(* IEC 61131-3 sources: std_i2980_v2.06_cp053/Source/IMM/ieccontrol/GlobalBaseArchives (part 20) *)

(* ---- ABUpdateRelLintabPreInject.pu ---- *)
IMPORT_OVER_LISTFILE
 FFixCylinderData
, FCalculateCylinderSize
, FCalcScrewSize
, KAPPL_LintabData
, tsCylinderData
, FBDebugTrace

END_IMPORT

ALGORITHM_BLOCK ABUpdateRelLintabPreInject #DUMMY_EDIT_BLOCK

SYSTEM_VAR
 sv_bCalcMaxValuesFromCylData : BOOL (* TRUE: calculate max speed and max pressure values by using cylinder data;  FALSE: max values must be entered manually *);
END_VAR

SYSTEM_OBJECT
 PU_Task_7 : TASK;
END_OBJECT

VAR
 mpLintabOut : REFTO KAPPL_LintabData;
 mpCylinderData : REFTO tsCylinderData;
 mprMaxPressure : REFTO REAL;
 mprMaxHydrPressure : REFTO REAL;
 mbInitDone : BOOL;
 mprScrewDiameter : REFTO REAL;
END_VAR

ALGORITHM aUpdateLintabOut

#BEGIN_EDIT_BLOCK
(**************************************** WARNING ********************************************
 *** The KEBA Kemro K2 System including software is not intended for safety control tasks! ***
 ***                       For further information see Comment tab!                        ***
 *********************************************************************************************)

// save data to Pre lintab
// normally a 1:1 lintab
mpLintabOut^.LintabPoints.uNoOfPoints := 2;
mpLintabOut^.LintabPoints.Point[1].rX := 0.0;
mpLintabOut^.LintabPoints.Point[1].rY := 0.0;
mpLintabOut^.LintabPoints.Point[2].rX := mprMaxPressure^;
mpLintabOut^.LintabPoints.Point[2].rY := mprMaxHydrPressure^;

;#END_EDIT_BLOCK END_ALGORITHM

ALGORITHM aCalcMaxPressure

VAR_TEMP
 rCylinderSize : REAL (* size of cylinder im mm˛ *);
 rScrewSize : REAL (* size of screw in mm˛ *);
 tmp : BOOL;
END_VAR
#BEGIN_EDIT_BLOCK
(**************************************** WARNING ********************************************
 *** The KEBA Kemro K2 System including software is not intended for safety control tasks! ***
 ***                       For further information see Comment tab!                        ***
 *********************************************************************************************)

IF NOT sv_bCalcMaxValuesFromCylData THEN
   // no calculation necessary
   RETURN;
END_IF;

tmp := FFixCylinderData(mpCylinderData);

// sanity check
IF mprScrewDiameter^ <= 0.0 THEN
   mprScrewDiameter^ := 34.0;
END_IF;

rCylinderSize := FCalculateCylinderSize(CylinderData := mpCylinderData^, bSmallSize := mpCylinderData^.bUseSmallSize,bCalcHighPressSize := FALSE);

rScrewSize := FCalcScrewSize(mprScrewDiameter^);

// calculate pressure for screw
mprMaxPressure^ := mprMaxHydrPressure^ * rCylinderSize / rScrewSize;

;#END_EDIT_BLOCK END_ALGORITHM

ALGORITHM aInit

VAR_INPUT
 pLintabOut : REFTO KAPPL_LintabData;
 prMaxPressure : REFTO REAL (* reference to calculated max. pressure *);
 prMaxHydrPressure : REFTO REAL (* reference to max. possible hydraulic pressure (depends on used pumps(s)) *);
 pCylinderData : REFTO tsCylinderData;
 prScrewDiameter : REFTO REAL (* diameter of screw in mm *);
END_VAR

VAR
 fbDebugTrace : FBDebugTrace;
END_VAR
#BEGIN_EDIT_BLOCK
(**************************************** WARNING ********************************************
 *** The KEBA Kemro K2 System including software is not intended for safety control tasks! ***
 ***                       For further information see Comment tab!                        ***
 *********************************************************************************************)

mbInitDone := FALSE;
mpCylinderData := pCylinderData;
mpLintabOut := pLintabOut;
mprMaxPressure := prMaxPressure;
mprMaxHydrPressure := prMaxHydrPressure;
mprScrewDiameter := prScrewDiameter;

IF NOT CHECK_REF(pCylinderData^) THEN
   fbDebugTrace('pCylinderData not valid');
   RETURN;
END_IF;

IF (NOT CHECK_REF(prScrewDiameter^)) THEN
   fbDebugTrace('prScrewDiameter not valid');
   RETURN;
END_IF;

IF (NOT CHECK_REF(pLintabOut^)) THEN
   fbDebugTrace('pLintabOut not valid');
   RETURN;
END_IF;

IF (NOT CHECK_REF(prMaxPressure^)) THEN
   fbDebugTrace('prMaxPressure not valid');
   RETURN;
END_IF;

IF (NOT CHECK_REF(prMaxHydrPressure^)) THEN
   fbDebugTrace('prMaxHydrPressure not valid');
   RETURN;
END_IF;

// init successful
mbInitDone := TRUE;

aCalcMaxPressure();

aUpdateLintabOut();

;#END_EDIT_BLOCK END_ALGORITHM

POSTUPDATE_ALGORITHM pUpdatePressure ON PU_Task_7 WITH mprMaxHydrPressure^,mpCylinderData^,mprScrewDiameter^

#BEGIN_EDIT_BLOCK
(**************************************** WARNING ********************************************
 *** The KEBA Kemro K2 System including software is not intended for safety control tasks! ***
 ***                       For further information see Comment tab!                        ***
 *********************************************************************************************)

IF NOT mbInitDone THEN
    RETURN;
END_IF;

aCalcMaxPressure();

;#END_EDIT_BLOCK END_ALGORITHM

POSTUPDATE_ALGORITHM pUpdatePressureLintab ON PU_Task_7 WITH mprMaxHydrPressure^,mprMaxPressure^

#BEGIN_EDIT_BLOCK
(**************************************** WARNING ********************************************
 *** The KEBA Kemro K2 System including software is not intended for safety control tasks! ***
 ***                       For further information see Comment tab!                        ***
 *********************************************************************************************)

IF NOT mbInitDone THEN
    RETURN;
END_IF;

// update lintab
aUpdateLintabOut();

;#END_EDIT_BLOCK END_ALGORITHM

END_ALGORITHM_BLOCK

#END_OF_IEC_PART

@Puma @IecEditor 6 114 @Pou 25
@@@BEG_Comment@@@

@@@END_Comment@@@

@BEG_Contents

@BEG_Func
@RT(17)FuncTreeContainer
3
@Var @RT(16)FFixCylinderData @RT(0) @T @T @DERIVED 0 @F @RT(8)FUNCTION @F
@T
@BEG_Attrib
0 @RT(0) @RT(0)
@END_Attrib
1 1 @F @F @F @F

@Var @RT(22)FCalculateCylinderSize @RT(0) @T @T @DERIVED 0 @F @RT(8)FUNCTION @F
@T
@BEG_Attrib
0 @RT(0) @RT(0)
@END_Attrib
1 1 @F @F @F @F

@Var @RT(14)FCalcScrewSize @RT(0) @T @T @DERIVED 0 @F @RT(8)FUNCTION @F
@T
@BEG_Attrib
0 @RT(0) @RT(0)
@END_Attrib
1 1 @F @F @F @F

@END_Func

@BEG_Const
@RT(18)ConstTreeContainer
0
@END_Const

@BEG_Export

@BEG_Kind
@ALGORITHM_BLOCK @RT(26)ABUpdateRelLintabPreInject @STRUCTURED_TEXT
@RT(0) @RT(0) @RT(0)
@END_Kind

@BEG_Dcl
@RT(16)DclTreeContainer
8
@Var @RT(28)sv_bCalcMaxValuesFromCylData @RT(0) @T @F @DT @RT(4)BOOL @RT(0) @T @T @BASIC 0 @F
@F @F
@T
@BEG_Attrib
3 @RT(0) @RT(117)TRUE: calculate max speed and max pressure values by using cylinder data;  FALSE: max values must be entered manually @RT(0)
@END_Attrib
1 8 @F @F @F @F

@Var @RT(9)PU_Task_7 @RT(0) @T @F @DT @RT(4)TASK @RT(0) @T @T @BASIC 0 @F
@F @F
@T
@BEG_Attrib
3 @RT(0) @RT(0) @RT(0)
@END_Attrib
1 7 @F @F @F @F

@Var @RT(11)mpLintabOut @RT(0) @T @T @REFTO 0 @F @DERIVED 0 @T @T @DT @RT(16)KAPPL_LintabData @RT(0) @T @T @UNKNOWN 0 @F
@F @F
@T
@BEG_Attrib
3 @RT(0) @RT(0) @RT(0)
@END_Attrib
1 0 @F @F @F @F

@Var @RT(14)mpCylinderData @RT(0) @T @T @REFTO 0 @F @DERIVED 0 @T @T @DT @RT(14)tsCylinderData @RT(0) @T @T @UNKNOWN 0 @F
@F @F
@T
@BEG_Attrib
3 @RT(0) @RT(0) @RT(0)
@END_Attrib
1 0 @F @F @F @F

@Var @RT(14)mprMaxPressure @RT(0) @T @T @REFTO 0 @T @DT @RT(4)REAL @RT(0) @T @T @BASIC 0 @F
@F @F
@T
@BEG_Attrib
3 @RT(0) @RT(0) @RT(0)
@END_Attrib
1 0 @F @F @F @F

@Var @RT(18)mprMaxHydrPressure @RT(0) @T @T @REFTO 0 @T @DT @RT(4)REAL @RT(0) @T @T @BASIC 0 @F
@F @F
@T
@BEG_Attrib
3 @RT(0) @RT(0) @RT(0)
@END_Attrib
1 0 @F @F @F @F

@Var @RT(10)mbInitDone @RT(0) @T @F @DT @RT(4)BOOL @RT(0) @T @T @BASIC 0 @F
@F @F
@T
@BEG_Attrib
3 @RT(0) @RT(0) @RT(0)
@END_Attrib
1 0 @F @F @F @F

@Var @RT(16)mprScrewDiameter @RT(0) @T @T @REFTO 0 @T @DT @RT(4)REAL @RT(0) @T @T @BASIC 0 @F
@F @F
@T
@BEG_Attrib
3 @RT(0) @RT(0) @RT(0)
@END_Attrib
1 0 @F @F @F @F

@END_Dcl

@END_Export

@BEG_Body

5

@BEG_Export

@BEG_Algo
@ALGORITHM @RT(16)aUpdateLintabOut @STRUCTURED_TEXT
@RT(0) @RT(0) @RT(0) @F @F
@END_Algo

@BEG_Dcl
@RT(16)DclTreeContainer
0
@END_Dcl

@END_Export

@BEG_Export

@BEG_Algo
@ALGORITHM @RT(16)aCalcMaxPressure @STRUCTURED_TEXT
@RT(0) @RT(0) @RT(0) @F @F
@END_Algo

@BEG_Dcl
@RT(16)DclTreeContainer
3
@Var @RT(13)rCylinderSize @RT(0) @T @F @DT @RT(4)REAL @RT(0) @T @T @BASIC 0 @F
@F @F
@T
@BEG_Attrib
3 @RT(0) @RT(23)size of cylinder im mm˛ @RT(0)
@END_Attrib
1 4 @F @F @F @F

@Var @RT(10)rScrewSize @RT(0) @T @F @DT @RT(4)REAL @RT(0) @T @T @BASIC 0 @F
@F @F
@T
@BEG_Attrib
3 @RT(0) @RT(20)size of screw in mm˛ @RT(0)
@END_Attrib
1 4 @F @F @F @F

@Var @RT(3)tmp @RT(0) @T @F @DT @RT(4)BOOL @RT(0) @T @T @BASIC 0 @F
@F @F
@T
@BEG_Attrib
3 @RT(0) @RT(0) @RT(0)
@END_Attrib
1 4 @F @F @F @F

@END_Dcl

@END_Export

@BEG_Export

@BEG_Algo
@ALGORITHM @RT(5)aInit @STRUCTURED_TEXT
@RT(0) @RT(0) @RT(0) @F @F
@END_Algo

@BEG_Dcl
@RT(16)DclTreeContainer
6
@Var @RT(10)pLintabOut @RT(0) @T @T @REFTO 0 @F @DERIVED 0 @T @T @DT @RT(16)KAPPL_LintabData @RT(0) @T @T @UNKNOWN 0 @F
@F @F
@T
@BEG_Attrib
3 @RT(0) @RT(0) @RT(0)
@END_Attrib
1 1 @F @F @F @F

@Var @RT(13)prMaxPressure @RT(0) @T @T @REFTO 0 @T @DT @RT(4)REAL @RT(0) @T @T @BASIC 0 @F
@F @F
@T
@BEG_Attrib
3 @RT(0) @RT(37)reference to calculated max. pressure @RT(0)
@END_Attrib
1 1 @F @F @F @F

@Var @RT(17)prMaxHydrPressure @RT(0) @T @T @REFTO 0 @T @DT @RT(4)REAL @RT(0) @T @T @BASIC 0 @F
@F @F
@T
@BEG_Attrib
3 @RT(0) @RT(72)reference to max. possible hydraulic pressure (depends on used pumps(s)) @RT(0)
@END_Attrib
1 1 @F @F @F @F

@Var @RT(13)pCylinderData @RT(0) @T @T @REFTO 0 @F @DERIVED 0 @T @T @DT @RT(14)tsCylinderData @RT(0) @T @T @UNKNOWN 0 @F
@F @F
@T
@BEG_Attrib
3 @RT(0) @RT(0) @RT(0)
@END_Attrib
1 1 @F @F @F @F

@Var @RT(15)prScrewDiameter @RT(0) @T @T @REFTO 0 @T @DT @RT(4)REAL @RT(0) @T @T @BASIC 0 @F
@F @F
@T
@BEG_Attrib
3 @RT(0) @RT(23)diameter of screw in mm @RT(0)
@END_Attrib
1 1 @F @F @F @F

@Var @RT(12)fbDebugTrace @RT(0) @T @T @DERIVED 0 @F @RT(12)FBDebugTrace @F
@T
@BEG_Attrib
3 @RT(0) @RT(0) @RT(0)
@END_Attrib
1 0 @F @F @F @F

@END_Dcl

@END_Export

@BEG_Export

@BEG_Algo
@POSTUPDATE_ALGORITHM @RT(15)pUpdatePressure @STRUCTURED_TEXT
@RT(0) @RT(53)mprMaxHydrPressure^,mpCylinderData^,mprScrewDiameter^ @RT(9)PU_Task_7 @F @F
@END_Algo

@BEG_Dcl
@RT(16)DclTreeContainer
0
@END_Dcl

@END_Export

@BEG_Export

@BEG_Algo
@POSTUPDATE_ALGORITHM @RT(21)pUpdatePressureLintab @STRUCTURED_TEXT
@RT(0) @RT(35)mprMaxHydrPressure^,mprMaxPressure^ @RT(9)PU_Task_7 @F @F
@END_Algo

@BEG_Dcl
@RT(16)DclTreeContainer
0
@END_Dcl

@END_Export

@BEG_Body
@TL(13)
(**************************************** WARNING ********************************************
 *** The KEBA Kemro K2 System including software is not intended for safety control tasks! ***
 ***                       For further information see Comment tab!                        ***
 *********************************************************************************************)

// save data to Pre lintab
// normally a 1:1 lintab
mpLintabOut^.LintabPoints.uNoOfPoints := 2;
mpLintabOut^.LintabPoints.Point[1].rX := 0.0;
mpLintabOut^.LintabPoints.Point[1].rY := 0.0;
mpLintabOut^.LintabPoints.Point[2].rX := mprMaxPressure^;
mpLintabOut^.LintabPoints.Point[2].rY := mprMaxHydrPressure^;

@END_Body

@@@BEG_Comment@@@
@TL(0)

@@@END_Comment@@@

@BEG_Body
@TL(25)
(**************************************** WARNING ********************************************
 *** The KEBA Kemro K2 System including software is not intended for safety control tasks! ***
 ***                       For further information see Comment tab!                        ***
 *********************************************************************************************)

IF NOT sv_bCalcMaxValuesFromCylData THEN
   // no calculation necessary
   RETURN;
END_IF;

tmp := FFixCylinderData(mpCylinderData);

// sanity check
IF mprScrewDiameter^ <= 0.0 THEN
   mprScrewDiameter^ := 34.0;
END_IF;

rCylinderSize := FCalculateCylinderSize(CylinderData := mpCylinderData^, bSmallSize := mpCylinderData^.bUseSmallSize,bCalcHighPressSize := FALSE);

rScrewSize := FCalcScrewSize(mprScrewDiameter^);

// calculate pressure for screw
mprMaxPressure^ := mprMaxHydrPressure^ * rCylinderSize / rScrewSize;

@END_Body

@@@BEG_Comment@@@
@TL(0)

@@@END_Comment@@@

@BEG_Body
@TL(45)
(**************************************** WARNING ********************************************
 *** The KEBA Kemro K2 System including software is not intended for safety control tasks! ***
 ***                       For further information see Comment tab!                        ***
 *********************************************************************************************)

mbInitDone := FALSE;
mpCylinderData := pCylinderData;
mpLintabOut := pLintabOut;
mprMaxPressure := prMaxPressure;
mprMaxHydrPressure := prMaxHydrPressure;
mprScrewDiameter := prScrewDiameter;

IF NOT CHECK_REF(pCylinderData^) THEN
   fbDebugTrace('pCylinderData not valid');
   RETURN;
END_IF;

IF (NOT CHECK_REF(prScrewDiameter^)) THEN
   fbDebugTrace('prScrewDiameter not valid');
   RETURN;
END_IF;

IF (NOT CHECK_REF(pLintabOut^)) THEN
   fbDebugTrace('pLintabOut not valid');
   RETURN;
END_IF;

IF (NOT CHECK_REF(prMaxPressure^)) THEN
   fbDebugTrace('prMaxPressure not valid');
   RETURN;
END_IF;

IF (NOT CHECK_REF(prMaxHydrPressure^)) THEN
   fbDebugTrace('prMaxHydrPressure not valid');
   RETURN;
END_IF;

// init successful
mbInitDone := TRUE;

aCalcMaxPressure();

aUpdateLintabOut();

@END_Body

@@@BEG_Comment@@@
@TL(0)

@@@END_Comment@@@

@BEG_Body
@TL(11)
(**************************************** WARNING ********************************************
 *** The KEBA Kemro K2 System including software is not intended for safety control tasks! ***
 ***                       For further information see Comment tab!                        ***
 *********************************************************************************************)

IF NOT mbInitDone THEN
    RETURN;
END_IF;

aCalcMaxPressure();

@END_Body

@@@BEG_Comment@@@
@TL(0)

@@@END_Comment@@@

@BEG_Body
@TL(12)
(**************************************** WARNING ********************************************
 *** The KEBA Kemro K2 System including software is not intended for safety control tasks! ***
 ***                       For further information see Comment tab!                        ***
 *********************************************************************************************)

IF NOT mbInitDone THEN
    RETURN;
END_IF;

// update lintab
aUpdateLintabOut();

@END_Body

@@@BEG_Comment@@@
@TL(0)

@@@END_Comment@@@
@END_Body

@END_Contents

(* ---- ABUpdateRelLintabVel.pu ---- *)
IMPORT_OVER_LISTFILE
 FFixCylinderData
, FCalculateCylinderSize
, FScaleAndFloor
, tnDataState
, KAPPL_LintabData
, tsCylinderData

END_IMPORT

ALGORITHM_BLOCK ABUpdateRelLintabVel #DUMMY_EDIT_BLOCK

SYSTEM_VAR
 sv_bCalcMaxValuesFromCylData : BOOL (* TRUE: calculate max speed and max pressure values by using cylinder data;  FALSE: max values must be entered manually *);
 sv_DataState : tnDataState;
 sv_iReadMachineDataCount : UDINT;
END_VAR

SYSTEM_OBJECT
 PU_Task_7 : TASK;
 PU_Task_3 : TASK;
END_OBJECT

VAR
 mpLintabOut : REFTO KAPPL_LintabData (* OUT: velocity lintab of movement *);
 mprAbsFlow : REFTO REAL (* IN: maximum absolute flow in l/min *);
 mpCylinderData : REFTO tsCylinderData (* IN: cylinder data *);
 mprMaxSpeed : REFTO REAL (* IN/OUT: max speed of movement *);
 mprMaxSpeedCalc : REFTO REAL (* IN/OUT: max speed of movement (calculated) *);
 mprMaxSpeedCalib : REFTO REAL (* IN/OUT: max speed of movement (calculated) *);
 mbprMaxSpeedCalibLinked : BOOL := FALSE (* IN/OUT: max speed of movement (calculated) *);
 mprMaxSpeedReducePercent : REFTO REAL (* IN: percentage to reduce max speed *);
 miMaxSpeedDigitsToFloor : SINT := 0 (* IN: max speed digits to floor *);
 mbInitDone : BOOL;
 mbFwd : BOOL;
END_VAR

ALGORITHM aUpdateLintabOut

#BEGIN_EDIT_BLOCK
(**************************************** WARNING ********************************************
 *** The KEBA Kemro K2 System including software is not intended for safety control tasks! ***
 ***                       For further information see Comment tab!                        ***
 *********************************************************************************************)

// save data to Vel lintab
mpLintabOut^.LintabPoints.uNoOfPoints := 2;
mpLintabOut^.LintabPoints.Point[1].rX := 0.0;
mpLintabOut^.LintabPoints.Point[1].rY := 0.0;
mpLintabOut^.LintabPoints.Point[2].rX := mprMaxSpeedCalc^;
mpLintabOut^.LintabPoints.Point[2].rY := 100.0; // %

;#END_EDIT_BLOCK END_ALGORITHM

ALGORITHM aCalcMaxVelocity

VAR_TEMP
 tmp : BOOL;
END_VAR

VAR
 rMaxFlow : REAL (* maximum flow in mm^3/sec *);
 rSize : REAL;
 bSmallSize : BOOL;
 rScalePercent : REAL;
END_VAR
#BEGIN_EDIT_BLOCK
(**************************************** WARNING ********************************************
 *** The KEBA Kemro K2 System including software is not intended for safety control tasks! ***
 ***                       For further information see Comment tab!                        ***
 *********************************************************************************************)

IF NOT sv_bCalcMaxValuesFromCylData THEN
   // no calculation necessary
   RETURN;
END_IF;

tmp := FFixCylinderData(mpCylinderData);

// convert from l/min to mm^3/sec
rMaxFlow := mprAbsFlow^ * 100.0 *100.0 *100.0 / 60.0;

bSmallSize := mbFwd AND mpCylinderData^.bUseSmallSize OR
                 ((NOT mbFwd AND NOT mpCylinderData^.bUseSmallSize));

rSize := FCalculateCylinderSize(CylinderData := mpCylinderData^,
                                bSmallSize := bSmallSize,
                                bCalcHighPressSize := FALSE);
// mmł/s / mm˛ ->mm/s
mprMaxSpeedCalc^ := rMaxFlow / rSize;
IF ((mbInitDone AND sv_DataState = nReady) AND (mprMaxSpeed^ > mprMaxSpeedCalc^)) THEN
   // prevent recalculation on machine data load except if max. value exceeds custom value
   rScalePercent := 100.0;
   IF mprMaxSpeedReducePercent <> EMPTY THEN
      rScalePercent := 100.0 - mprMaxSpeedReducePercent^;
   END_IF;
   mprMaxSpeed^ := FScaleAndFloor(mprMaxSpeedCalc^, rScalePercent, miMaxSpeedDigitsToFloor);
END_IF;
// check max velocity for visualization
IF (mbprMaxSpeedCalibLinked) THEN
   IF(mprMaxSpeedCalib^ <= 0.0) OR (mprMaxSpeedCalib^ > mprMaxSpeedCalc^) THEN
      mprMaxSpeedCalib^ := mprMaxSpeedCalc^;
   END_IF;
END_IF;

;#END_EDIT_BLOCK END_ALGORITHM

ALGORITHM aInit

VAR_INPUT
 pLintabOut : REFTO KAPPL_LintabData;
 prMaxSpeed : REFTO REAL;
 prMaxSpeedCalc : REFTO REAL;
 prAbsFlow : REFTO REAL (* absolute flow in l/min *);
 bFwd : BOOL (* TRUE if block is used for fwd movement *);
 pCylinderData : REFTO tsCylinderData;
 prMaxSpeedReducePercent : REFTO REAL;
 iMaxSpeedDigitsToFloor : SINT;
 prMaxSpeedCalib : REFTO REAL;
END_VAR

VAR
 // prMaxPumpFlow : REFTO REAL;
 tmp : DINT;
END_VAR
#BEGIN_EDIT_BLOCK
(**************************************** WARNING ********************************************
 *** The KEBA Kemro K2 System including software is not intended for safety control tasks! ***
 ***                       For further information see Comment tab!                        ***
 *********************************************************************************************)

mbInitDone := FALSE;
mprAbsFlow := prAbsFlow;
mpCylinderData := pCylinderData;
mpLintabOut := pLintabOut;
mprMaxSpeed := prMaxSpeed;
mprMaxSpeedCalc := prMaxSpeedCalc;
mprMaxSpeedCalib := prMaxSpeedCalib;
mprMaxSpeedReducePercent := prMaxSpeedReducePercent;
miMaxSpeedDigitsToFloor := iMaxSpeedDigitsToFloor;
mbFwd := bFwd;

IF NOT CHECK_REF(prAbsFlow^) THEN
    tmp := Print('prAbsFlow not valid');
    RETURN;
END_IF;

IF NOT CHECK_REF(pCylinderData^) THEN
    tmp := Print('pCylinderData not valid');
    RETURN;
END_IF;

IF (NOT CHECK_REF(pLintabOut^)) THEN
    tmp := Print('pLintabOut not valid');
    RETURN;
END_IF;

IF (NOT CHECK_REF(prMaxSpeed^)) THEN
    tmp := Print('prMaxSpeed not valid');
    RETURN;
END_IF;

IF (NOT CHECK_REF(prMaxSpeedCalc^)) THEN
    tmp := Print('prMaxSpeedCalc not valid');
    RETURN;
END_IF;

IF (CHECK_REF(mprMaxSpeedCalib^)) THEN
    mbprMaxSpeedCalibLinked := TRUE;
END_IF;

aCalcMaxVelocity();

//update lintab
aUpdateLintabOut();

// init successful
mbInitDone := TRUE;

;#END_EDIT_BLOCK END_ALGORITHM

POSTUPDATE_ALGORITHM pUpdateVelocity ON PU_Task_7 WITH mprAbsFlow^,mpCylinderData^

#BEGIN_EDIT_BLOCK
(**************************************** WARNING ********************************************
 *** The KEBA Kemro K2 System including software is not intended for safety control tasks! ***
 ***                       For further information see Comment tab!                        ***
 *********************************************************************************************)

IF NOT mbInitDone OR (sv_DataState = nReadMachineData) THEN
   RETURN;
END_IF;

// reset calib value if diameter or flow is changed
IF mbprMaxSpeedCalibLinked AND (sv_DataState = nReady) THEN
   mprMaxSpeedCalib^ := 0.0;
END_IF;

aCalcMaxVelocity();

;#END_EDIT_BLOCK END_ALGORITHM

POSTUPDATE_ALGORITHM pUpdateVelocityLintab ON PU_Task_7 WITH mprMaxSpeedCalc^

#BEGIN_EDIT_BLOCK
(**************************************** WARNING ********************************************
 *** The KEBA Kemro K2 System including software is not intended for safety control tasks! ***
 ***                       For further information see Comment tab!                        ***
 *********************************************************************************************)

IF NOT mbInitDone THEN
    RETURN;
END_IF;

aUpdateLintabOut();

;#END_EDIT_BLOCK END_ALGORITHM

POSTUPDATE_ALGORITHM pUpdateMaxVelocity ON PU_Task_7 WITH mprMaxSpeedCalib^

VAR
 rScalePercent : REAL;
END_VAR
#BEGIN_EDIT_BLOCK
(**************************************** WARNING ********************************************
 *** The KEBA Kemro K2 System including software is not intended for safety control tasks! ***
 ***                       For further information see Comment tab!                        ***
 *********************************************************************************************)

IF sv_DataState = nReadMachineData THEN
   RETURN;
END_IF;

IF ((mprMaxSpeedCalib^ < mprMaxSpeed^) AND (mprMaxSpeedCalib^ > 0.0)) THEN
   rScalePercent := 100.0;
   IF mprMaxSpeedReducePercent <> EMPTY THEN
      rScalePercent := 100.0 - mprMaxSpeedReducePercent^;
   END_IF;
   mprMaxSpeed^ := FScaleAndFloor(mprMaxSpeedCalib^, rScalePercent, miMaxSpeedDigitsToFloor);
END_IF;

;#END_EDIT_BLOCK END_ALGORITHM

POSTUPDATE_ALGORITHM pMachineDataLoaded ON PU_Task_7 WITH sv_iReadMachineDataCount

#BEGIN_EDIT_BLOCK
(**************************************** WARNING ********************************************
 *** The KEBA Kemro K2 System including software is not intended for safety control tasks! ***
 ***                       For further information see Comment tab!                        ***
 *********************************************************************************************)

aCalcMaxVelocity();

;#END_EDIT_BLOCK END_ALGORITHM

POSTUPDATE_ALGORITHM pMachineDataLoadingStarted ON PU_Task_3(1) WITH sv_DataState

#BEGIN_EDIT_BLOCK
(**************************************** WARNING ********************************************
 *** The KEBA Kemro K2 System including software is not intended for safety control tasks! ***
 ***                       For further information see Comment tab!                        ***
 *********************************************************************************************)

IF sv_DataState = nReadMachineData THEN
   //reset max speed calib at the beginning of machine data loading
   //if max speed calib is part of the loaded machine data, the correct value comes from the XMl file
   //if max speed calib is not part of machine data it is set to max speed calc
   //when calling aCalcMaxVelocity after loading machine data is finished
   IF mbprMaxSpeedCalibLinked THEN
      mprMaxSpeedCalib^ := 0.0;
   END_IF;
END_IF;

;#END_EDIT_BLOCK END_ALGORITHM

END_ALGORITHM_BLOCK

#END_OF_IEC_PART

@Puma @IecEditor 6 114 @Pou 25
@@@BEG_Comment@@@

@@@END_Comment@@@

@BEG_Contents

@BEG_Func
@RT(17)FuncTreeContainer
3
@Var @RT(16)FFixCylinderData @RT(0) @T @T @DERIVED 0 @F @RT(8)FUNCTION @F
@T
@BEG_Attrib
0 @RT(0) @RT(0)
@END_Attrib
1 1 @F @F @F @F

@Var @RT(22)FCalculateCylinderSize @RT(0) @T @T @DERIVED 0 @F @RT(8)FUNCTION @F
@T
@BEG_Attrib
0 @RT(0) @RT(0)
@END_Attrib
1 1 @F @F @F @F

@Var @RT(14)FScaleAndFloor @RT(0) @T @T @DERIVED 0 @F @RT(8)FUNCTION @F
@T
@BEG_Attrib
0 @RT(0) @RT(0)
@END_Attrib
1 1 @F @F @F @F

@END_Func

@BEG_Const
@RT(18)ConstTreeContainer
0
@END_Const

@BEG_Export

@BEG_Kind
@ALGORITHM_BLOCK @RT(20)ABUpdateRelLintabVel @STRUCTURED_TEXT
@RT(0) @RT(0) @RT(0)
@END_Kind

@BEG_Dcl
@RT(16)DclTreeContainer
16
@Var @RT(28)sv_bCalcMaxValuesFromCylData @RT(0) @T @F @DT @RT(4)BOOL @RT(0) @T @T @BASIC 0 @F
@F @F
@T
@BEG_Attrib
3 @RT(0) @RT(117)TRUE: calculate max speed and max pressure values by using cylinder data;  FALSE: max values must be entered manually @RT(0)
@END_Attrib
1 8 @F @F @F @F

@Var @RT(12)sv_DataState @RT(0) @T @T @DERIVED 0 @T @T @DT @RT(11)tnDataState @RT(0) @T @T @UNKNOWN 0 @F
@F @F
@T
@BEG_Attrib
3 @RT(0) @RT(0) @RT(0)
@END_Attrib
1 8 @F @F @F @F

@Var @RT(9)PU_Task_7 @RT(0) @T @F @DT @RT(4)TASK @RT(0) @T @T @BASIC 0 @F
@F @F
@T
@BEG_Attrib
3 @RT(0) @RT(0) @RT(0)
@END_Attrib
1 7 @F @F @F @F

@Var @RT(11)mpLintabOut @RT(0) @T @T @REFTO 0 @F @DERIVED 0 @T @T @DT @RT(16)KAPPL_LintabData @RT(0) @T @T @UNKNOWN 0 @F
@F @F
@T
@BEG_Attrib
3 @RT(0) @RT(32)OUT: velocity lintab of movement @RT(0)
@END_Attrib
1 0 @F @F @F @F

@Var @RT(10)mprAbsFlow @RT(0) @T @T @REFTO 0 @T @DT @RT(4)REAL @RT(0) @T @T @BASIC 0 @F
@F @F
@T
@BEG_Attrib
3 @RT(0) @RT(34)IN: maximum absolute flow in l/min @RT(0)
@END_Attrib
1 0 @F @F @F @F

@Var @RT(14)mpCylinderData @RT(0) @T @T @REFTO 0 @F @DERIVED 0 @T @T @DT @RT(14)tsCylinderData @RT(0) @T @T @UNKNOWN 0 @F
@F @F
@T
@BEG_Attrib
3 @RT(0) @RT(17)IN: cylinder data @RT(0)
@END_Attrib
1 0 @F @F @F @F

@Var @RT(11)mprMaxSpeed @RT(0) @T @T @REFTO 0 @T @DT @RT(4)REAL @RT(0) @T @T @BASIC 0 @F
@F @F
@T
@BEG_Attrib
3 @RT(0) @RT(29)IN/OUT: max speed of movement @RT(0)
@END_Attrib
1 0 @F @F @F @F

@Var @RT(15)mprMaxSpeedCalc @RT(0) @T @T @REFTO 0 @T @DT @RT(4)REAL @RT(0) @T @T @BASIC 0 @F
@F @F
@T
@BEG_Attrib
3 @RT(0) @RT(42)IN/OUT: max speed of movement (calculated) @RT(0)
@END_Attrib
1 0 @F @F @F @F

@Var @RT(16)mprMaxSpeedCalib @RT(0) @T @T @REFTO 0 @T @DT @RT(4)REAL @RT(0) @T @T @BASIC 0 @F
@F @F
@T
@BEG_Attrib
3 @RT(0) @RT(42)IN/OUT: max speed of movement (calculated) @RT(0)
@END_Attrib
1 0 @F @F @F @F

@Var @RT(23)mbprMaxSpeedCalibLinked @RT(0) @T @F @DT @RT(4)BOOL @RT(0) @T @T @BASIC 0 @F
@F @F
@T
@BEG_Attrib
3 @RT(5)FALSE @RT(42)IN/OUT: max speed of movement (calculated) @RT(0)
@END_Attrib
1 0 @F @F @F @F

@Var @RT(24)mprMaxSpeedReducePercent @RT(0) @T @T @REFTO 0 @T @DT @RT(4)REAL @RT(0) @T @T @BASIC 0 @F
@F @F
@T
@BEG_Attrib
3 @RT(0) @RT(34)IN: percentage to reduce max speed @RT(0)
@END_Attrib
1 0 @F @F @F @F

@Var @RT(23)miMaxSpeedDigitsToFloor @RT(0) @T @F @DT @RT(4)SINT @RT(0) @T @T @BASIC 0 @F
@F @F
@T
@BEG_Attrib
3 @RT(1)0 @RT(29)IN: max speed digits to floor @RT(0)
@END_Attrib
1 0 @F @F @F @F

@Var @RT(10)mbInitDone @RT(0) @T @F @DT @RT(4)BOOL @RT(0) @T @T @BASIC 0 @F
@F @F
@T
@BEG_Attrib
3 @RT(0) @RT(0) @RT(0)
@END_Attrib
1 0 @F @F @F @F

@Var @RT(5)mbFwd @RT(0) @T @F @DT @RT(4)BOOL @RT(0) @T @T @BASIC 0 @F
@F @F
@T
@BEG_Attrib
3 @RT(0) @RT(0) @RT(0)
@END_Attrib
1 0 @F @F @F @F

@Var @RT(24)sv_iReadMachineDataCount @RT(0) @T @T @RENAMED 0 @T @T @DT @RT(5)UDINT @RT(0) @T @T @BASIC 0 @F
@F @F
@T
@BEG_Attrib
3 @RT(0) @RT(0) @RT(0)
@END_Attrib
1 8 @F @F @F @F

@Var @RT(9)PU_Task_3 @RT(0) @T @T @RENAMED 0 @T @T @DT @RT(4)TASK @RT(0) @T @T @BASIC 0 @F
@F @F
@T
@BEG_Attrib
3 @RT(0) @RT(0) @RT(0)
@END_Attrib
1 7 @F @F @F @F

@END_Dcl

@END_Export

@BEG_Body

8

@BEG_Export

@BEG_Algo
@ALGORITHM @RT(16)aUpdateLintabOut @STRUCTURED_TEXT
@RT(0) @RT(0) @RT(0) @F @F
@END_Algo

@BEG_Dcl
@RT(16)DclTreeContainer
0
@END_Dcl

@END_Export

@BEG_Export

@BEG_Algo
@ALGORITHM @RT(16)aCalcMaxVelocity @STRUCTURED_TEXT
@RT(0) @RT(0) @RT(0) @F @F
@END_Algo

@BEG_Dcl
@RT(16)DclTreeContainer
5
@Var @RT(3)tmp @RT(0) @T @F @DT @RT(4)BOOL @RT(0) @T @T @BASIC 0 @F
@F @F
@T
@BEG_Attrib
3 @RT(0) @RT(0) @RT(0)
@END_Attrib
1 4 @F @F @F @F

@Var @RT(8)rMaxFlow @RT(0) @T @F @DT @RT(4)REAL @RT(0) @T @T @BASIC 0 @F
@F @F
@T
@BEG_Attrib
3 @RT(0) @RT(24)maximum flow in mm^3/sec @RT(0)
@END_Attrib
1 0 @F @F @F @F

@Var @RT(5)rSize @RT(0) @T @F @DT @RT(4)REAL @RT(0) @T @T @BASIC 0 @F
@F @F
@T
@BEG_Attrib
3 @RT(0) @RT(0) @RT(0)
@END_Attrib
1 0 @F @F @F @F

@Var @RT(10)bSmallSize @RT(0) @T @F @DT @RT(4)BOOL @RT(0) @T @T @BASIC 0 @F
@F @F
@T
@BEG_Attrib
3 @RT(0) @RT(0) @RT(0)
@END_Attrib
1 0 @F @F @F @F

@Var @RT(13)rScalePercent @RT(0) @T @F @DT @RT(4)REAL @RT(0) @T @T @BASIC 0 @F
@F @F
@T
@BEG_Attrib
3 @RT(0) @RT(0) @RT(0)
@END_Attrib
1 0 @F @F @F @F

@END_Dcl

@END_Export

@BEG_Export

@BEG_Algo
@ALGORITHM @RT(5)aInit @STRUCTURED_TEXT
@RT(0) @RT(0) @RT(0) @F @F
@END_Algo

@BEG_Dcl
@RT(16)DclTreeContainer
11
@Var @RT(10)pLintabOut @RT(0) @T @T @REFTO 0 @F @DERIVED 0 @T @T @DT @RT(16)KAPPL_LintabData @RT(0) @T @T @UNKNOWN 0 @F
@F @F
@T
@BEG_Attrib
3 @RT(0) @RT(0) @RT(0)
@END_Attrib
1 1 @F @F @F @F

@Var @RT(10)prMaxSpeed @RT(0) @T @T @REFTO 0 @T @DT @RT(4)REAL @RT(0) @T @T @BASIC 0 @F
@F @F
@T
@BEG_Attrib
3 @RT(0) @RT(0) @RT(0)
@END_Attrib
1 1 @F @F @F @F

@Var @RT(14)prMaxSpeedCalc @RT(0) @T @T @REFTO 0 @T @DT @RT(4)REAL @RT(0) @T @T @BASIC 0 @F
@F @F
@T
@BEG_Attrib
3 @RT(0) @RT(0) @RT(0)
@END_Attrib
1 1 @F @F @F @F

@Var @RT(9)prAbsFlow @RT(0) @T @T @REFTO 0 @T @DT @RT(4)REAL @RT(0) @T @T @BASIC 0 @F
@F @F
@T
@BEG_Attrib
3 @RT(0) @RT(22)absolute flow in l/min @RT(0)
@END_Attrib
1 1 @F @F @F @F

@Var @RT(4)bFwd @RT(0) @T @F @DT @RT(4)BOOL @RT(0) @T @T @BASIC 0 @F
@F @F
@T
@BEG_Attrib
3 @RT(0) @RT(38)TRUE if block is used for fwd movement @RT(0)
@END_Attrib
1 1 @F @F @F @F

@Var @RT(13)pCylinderData @RT(0) @T @T @REFTO 0 @F @DERIVED 0 @T @T @DT @RT(14)tsCylinderData @RT(0) @T @T @UNKNOWN 0 @F
@F @F
@T
@BEG_Attrib
3 @RT(0) @RT(0) @RT(0)
@END_Attrib
1 1 @F @F @F @F

@Var @RT(23)prMaxSpeedReducePercent @RT(0) @T @T @REFTO 0 @T @DT @RT(4)REAL @RT(0) @T @T @BASIC 0 @F
@F @F
@T
@BEG_Attrib
3 @RT(0) @RT(0) @RT(0)
@END_Attrib
1 1 @F @F @F @F

@Var @RT(22)iMaxSpeedDigitsToFloor @RT(0) @T @F @DT @RT(4)SINT @RT(0) @T @T @BASIC 0 @F
@F @F
@T
@BEG_Attrib
3 @RT(0) @RT(0) @RT(0)
@END_Attrib
1 1 @F @F @F @F

@Var @RT(13)prMaxPumpFlow @RT(0) @T @T @REFTO 0 @T @DT @RT(4)REAL @RT(0) @T @T @BASIC 0 @F
@F @T
@T
@BEG_Attrib
3 @RT(0) @RT(0) @RT(0)
@END_Attrib
1 0 @F @F @F @F

@Var @RT(3)tmp @RT(0) @T @F @DT @RT(4)DINT @RT(0) @T @T @BASIC 0 @F
@F @F
@T
@BEG_Attrib
3 @RT(0) @RT(0) @RT(0)
@END_Attrib
1 0 @F @F @F @F

@Var @RT(15)prMaxSpeedCalib @RT(0) @T @T @REFTO 0 @T @DT @RT(4)REAL @RT(0) @T @T @BASIC 0 @F
@F @F
@T
@BEG_Attrib
3 @RT(0) @RT(0) @RT(0)
@END_Attrib
1 1 @F @F @F @F

@END_Dcl

@END_Export

@BEG_Export

@BEG_Algo
@POSTUPDATE_ALGORITHM @RT(15)pUpdateVelocity @STRUCTURED_TEXT
@RT(0) @RT(27)mprAbsFlow^,mpCylinderData^ @RT(9)PU_Task_7 @F @F
@END_Algo

@BEG_Dcl
@RT(16)DclTreeContainer
0
@END_Dcl

@END_Export

@BEG_Export

@BEG_Algo
@POSTUPDATE_ALGORITHM @RT(21)pUpdateVelocityLintab @STRUCTURED_TEXT
@RT(0) @RT(16)mprMaxSpeedCalc^ @RT(9)PU_Task_7 @F @F
@END_Algo

@BEG_Dcl
@RT(16)DclTreeContainer
0
@END_Dcl

@END_Export

@BEG_Export

@BEG_Algo
@POSTUPDATE_ALGORITHM @RT(18)pUpdateMaxVelocity @STRUCTURED_TEXT
@RT(0) @RT(17)mprMaxSpeedCalib^ @RT(9)PU_Task_7 @F @F
@END_Algo

@BEG_Dcl
@RT(16)DclTreeContainer
1
@Var @RT(13)rScalePercent @RT(0) @T @F @DT @RT(4)REAL @RT(0) @T @T @BASIC 0 @F
@F @F
@T
@BEG_Attrib
3 @RT(0) @RT(0) @RT(0)
@END_Attrib
1 0 @F @F @F @F

@END_Dcl

@END_Export

@BEG_Export

@BEG_Algo
@POSTUPDATE_ALGORITHM @RT(18)pMachineDataLoaded @STRUCTURED_TEXT
@RT(0) @RT(24)sv_iReadMachineDataCount @RT(9)PU_Task_7 @F @F
@END_Algo

@BEG_Dcl
@RT(16)DclTreeContainer
0
@END_Dcl

@END_Export

@BEG_Export

@BEG_Algo
@POSTUPDATE_ALGORITHM @RT(26)pMachineDataLoadingStarted @STRUCTURED_TEXT
@RT(0) @RT(12)sv_DataState @RT(12)PU_Task_3(1) @F @F
@END_Algo

@BEG_Dcl
@RT(16)DclTreeContainer
0
@END_Dcl

@END_Export

@BEG_Body
@TL(12)
(**************************************** WARNING ********************************************
 *** The KEBA Kemro K2 System including software is not intended for safety control tasks! ***
 ***                       For further information see Comment tab!                        ***
 *********************************************************************************************)

// save data to Vel lintab
mpLintabOut^.LintabPoints.uNoOfPoints := 2;
mpLintabOut^.LintabPoints.Point[1].rX := 0.0;
mpLintabOut^.LintabPoints.Point[1].rY := 0.0;
mpLintabOut^.LintabPoints.Point[2].rX := mprMaxSpeedCalc^;
mpLintabOut^.LintabPoints.Point[2].rY := 100.0; // %

@END_Body

@@@BEG_Comment@@@
@TL(0)

@@@END_Comment@@@

@BEG_Body
@TL(42)
(**************************************** WARNING ********************************************
 *** The KEBA Kemro K2 System including software is not intended for safety control tasks! ***
 ***                       For further information see Comment tab!                        ***
 *********************************************************************************************)

IF NOT sv_bCalcMaxValuesFromCylData THEN
   // no calculation necessary
   RETURN;
END_IF;

tmp := FFixCylinderData(mpCylinderData);

// convert from l/min to mm^3/sec
rMaxFlow := mprAbsFlow^ * 100.0 *100.0 *100.0 / 60.0;

bSmallSize := mbFwd AND mpCylinderData^.bUseSmallSize OR
                 ((NOT mbFwd AND NOT mpCylinderData^.bUseSmallSize));

rSize := FCalculateCylinderSize(CylinderData := mpCylinderData^,
                                bSmallSize := bSmallSize,
                                bCalcHighPressSize := FALSE);
// mmł/s / mm˛ ->mm/s
mprMaxSpeedCalc^ := rMaxFlow / rSize;
IF ((mbInitDone AND sv_DataState = nReady) AND (mprMaxSpeed^ > mprMaxSpeedCalc^)) THEN
   // prevent recalculation on machine data load except if max. value exceeds custom value
   rScalePercent := 100.0;
   IF mprMaxSpeedReducePercent <> EMPTY THEN
      rScalePercent := 100.0 - mprMaxSpeedReducePercent^;
   END_IF;
   mprMaxSpeed^ := FScaleAndFloor(mprMaxSpeedCalc^, rScalePercent, miMaxSpeedDigitsToFloor);
END_IF;
// check max velocity for visualization
IF (mbprMaxSpeedCalibLinked) THEN
   IF(mprMaxSpeedCalib^ <= 0.0) OR (mprMaxSpeedCalib^ > mprMaxSpeedCalc^) THEN
      mprMaxSpeedCalib^ := mprMaxSpeedCalc^;
   END_IF;
END_IF;

@END_Body

@@@BEG_Comment@@@
@TL(0)

@@@END_Comment@@@

@BEG_Body
@TL(54)
(**************************************** WARNING ********************************************
 *** The KEBA Kemro K2 System including software is not intended for safety control tasks! ***
 ***                       For further information see Comment tab!                        ***
 *********************************************************************************************)

mbInitDone := FALSE;
mprAbsFlow := prAbsFlow;
mpCylinderData := pCylinderData;
mpLintabOut := pLintabOut;
mprMaxSpeed := prMaxSpeed;
mprMaxSpeedCalc := prMaxSpeedCalc;
mprMaxSpeedCalib := prMaxSpeedCalib;
mprMaxSpeedReducePercent := prMaxSpeedReducePercent;
miMaxSpeedDigitsToFloor := iMaxSpeedDigitsToFloor;
mbFwd := bFwd;

IF NOT CHECK_REF(prAbsFlow^) THEN
    tmp := Print('prAbsFlow not valid');
    RETURN;
END_IF;

IF NOT CHECK_REF(pCylinderData^) THEN
    tmp := Print('pCylinderData not valid');
    RETURN;
END_IF;

IF (NOT CHECK_REF(pLintabOut^)) THEN
    tmp := Print('pLintabOut not valid');
    RETURN;
END_IF;

IF (NOT CHECK_REF(prMaxSpeed^)) THEN
    tmp := Print('prMaxSpeed not valid');
    RETURN;
END_IF;

IF (NOT CHECK_REF(prMaxSpeedCalc^)) THEN
    tmp := Print('prMaxSpeedCalc not valid');
    RETURN;
END_IF;

IF (CHECK_REF(mprMaxSpeedCalib^)) THEN
    mbprMaxSpeedCalibLinked := TRUE;
END_IF;

aCalcMaxVelocity();

//update lintab
aUpdateLintabOut();

// init successful
mbInitDone := TRUE;

@END_Body

@@@BEG_Comment@@@
@TL(0)

@@@END_Comment@@@

@BEG_Body
@TL(20)
(**************************************** WARNING ********************************************
 *** The KEBA Kemro K2 System including software is not intended for safety control tasks! ***
 ***                       For further information see Comment tab!                        ***
 *********************************************************************************************)

IF NOT mbInitDone OR (sv_DataState = nReadMachineData) THEN
   RETURN;
END_IF;

// reset calib value if diameter or flow is changed
IF mbprMaxSpeedCalibLinked AND (sv_DataState = nReady) THEN
   mprMaxSpeedCalib^ := 0.0;
END_IF;

aCalcMaxVelocity();

@END_Body

@@@BEG_Comment@@@
@TL(0)

@@@END_Comment@@@

@BEG_Body
@TL(13)
(**************************************** WARNING ********************************************
 *** The KEBA Kemro K2 System including software is not intended for safety control tasks! ***
 ***                       For further information see Comment tab!                        ***
 *********************************************************************************************)

IF NOT mbInitDone THEN
    RETURN;
END_IF;

aUpdateLintabOut();

@END_Body

@@@BEG_Comment@@@
@TL(0)

@@@END_Comment@@@

@BEG_Body
@TL(18)
(**************************************** WARNING ********************************************
 *** The KEBA Kemro K2 System including software is not intended for safety control tasks! ***
 ***                       For further information see Comment tab!                        ***
 *********************************************************************************************)

IF sv_DataState = nReadMachineData THEN
   RETURN;
END_IF;

IF ((mprMaxSpeedCalib^ < mprMaxSpeed^) AND (mprMaxSpeedCalib^ > 0.0)) THEN
   rScalePercent := 100.0;
   IF mprMaxSpeedReducePercent <> EMPTY THEN
      rScalePercent := 100.0 - mprMaxSpeedReducePercent^;
   END_IF;
   mprMaxSpeed^ := FScaleAndFloor(mprMaxSpeedCalib^, rScalePercent, miMaxSpeedDigitsToFloor);
END_IF;

@END_Body

@@@BEG_Comment@@@
@TL(0)

@@@END_Comment@@@

@BEG_Body
@TL(7)
(**************************************** WARNING ********************************************
 *** The KEBA Kemro K2 System including software is not intended for safety control tasks! ***
 ***                       For further information see Comment tab!                        ***
 *********************************************************************************************)

aCalcMaxVelocity();

@END_Body

@@@BEG_Comment@@@
@TL(0)

@@@END_Comment@@@

@BEG_Body
@TL(15)
(**************************************** WARNING ********************************************
 *** The KEBA Kemro K2 System including software is not intended for safety control tasks! ***
 ***                       For further information see Comment tab!                        ***
 *********************************************************************************************)

IF sv_DataState = nReadMachineData THEN
   //reset max speed calib at the beginning of machine data loading
   //if max speed calib is part of the loaded machine data, the correct value comes from the XMl file
   //if max speed calib is not part of machine data it is set to max speed calc
   //when calling aCalcMaxVelocity after loading machine data is finished
   IF mbprMaxSpeedCalibLinked THEN
      mprMaxSpeedCalib^ := 0.0;
   END_IF;
END_IF;

@END_Body

@@@BEG_Comment@@@
@TL(0)

@@@END_Comment@@@
@END_Body

@END_Contents

(* ---- ABUpdateRelLintabVelCore.pu ---- *)
IMPORT_OVER_LISTFILE
 KAPPL_LintabData

END_IMPORT

ALGORITHM_BLOCK ABUpdateRelLintabVelCore #DUMMY_EDIT_BLOCK

SYSTEM_VAR
 sv_bCalcMaxValuesFromCylData : BOOL (* TRUE: calculate max speed and max pressure values by using cylinder data;  FALSE: max values must be entered manually *);
END_VAR

SYSTEM_OBJECT
 PU_Task_7 : TASK;
END_OBJECT

VAR
 mpLintabOut : REFTO KAPPL_LintabData (* OUT: velocity lintab of movement *);
 mprAbsFlow : REFTO REAL (* IN: maximum absolute flow in l/min *);
 mprMaxSpeed : REFTO REAL (* IN/OUT: max speed of fwd movement *);
 mbInitDone : BOOL;
END_VAR

ALGORITHM aUpdateLintabOut

#BEGIN_EDIT_BLOCK
(**************************************** WARNING ********************************************
 *** The KEBA Kemro K2 System including software is not intended for safety control tasks! ***
 ***                       For further information see Comment tab!                        ***
 *********************************************************************************************)

// save data to Vel lintab
mpLintabOut^.LintabPoints.uNoOfPoints := 2;
mpLintabOut^.LintabPoints.Point[1].rX := 0.0;
mpLintabOut^.LintabPoints.Point[1].rY := 0.0;
mpLintabOut^.LintabPoints.Point[2].rX := mprMaxSpeed^;
mpLintabOut^.LintabPoints.Point[2].rY := 100.0; // %

;#END_EDIT_BLOCK END_ALGORITHM

ALGORITHM aCalcMaxSpeed

#BEGIN_EDIT_BLOCK
(**************************************** WARNING ********************************************
 *** The KEBA Kemro K2 System including software is not intended for safety control tasks! ***
 ***                       For further information see Comment tab!                        ***
 *********************************************************************************************)

IF NOT sv_bCalcMaxValuesFromCylData THEN
   // no calculation necessary
   RETURN;
END_IF;

// max flow in l/min
mprMaxSpeed^ := mprAbsFlow^;

;#END_EDIT_BLOCK END_ALGORITHM

ALGORITHM aInit

VAR_INPUT
 pLintabOut : REFTO KAPPL_LintabData;
 prMaxSpeed : REFTO REAL;
 prAbsFlow : REFTO REAL (* absolute flow in l/min *);
END_VAR

VAR
 tmp : DINT;
END_VAR
#BEGIN_EDIT_BLOCK
(**************************************** WARNING ********************************************
 *** The KEBA Kemro K2 System including software is not intended for safety control tasks! ***
 ***                       For further information see Comment tab!                        ***
 *********************************************************************************************)

mbInitDone := FALSE;
mprAbsFlow := prAbsFlow;
mpLintabOut := pLintabOut;
mprMaxSpeed := prMaxSpeed;

IF NOT CHECK_REF(prAbsFlow^) THEN
    tmp := Print('prAbsFlow not valid');
    RETURN;
END_IF;

IF (NOT CHECK_REF(pLintabOut^)) THEN
    tmp := Print('pLintabOut not valid');
    RETURN;
END_IF;

IF (NOT CHECK_REF(prMaxSpeed^)) THEN
    tmp := Print('prMaxSpeed not valid');
    RETURN;
END_IF;

// init successful
mbInitDone := TRUE;

aCalcMaxSpeed();

aUpdateLintabOut();

;#END_EDIT_BLOCK END_ALGORITHM

POSTUPDATE_ALGORITHM pUpdateVelocity ON PU_Task_7 WITH mprAbsFlow^

#BEGIN_EDIT_BLOCK
(**************************************** WARNING ********************************************
 *** The KEBA Kemro K2 System including software is not intended for safety control tasks! ***
 ***                       For further information see Comment tab!                        ***
 *********************************************************************************************)

IF NOT mbInitDone THEN
    RETURN;
END_IF;

aCalcMaxSpeed();

;#END_EDIT_BLOCK END_ALGORITHM

POSTUPDATE_ALGORITHM pUpdateVelocityLintab ON PU_Task_7 WITH mprMaxSpeed^

#BEGIN_EDIT_BLOCK
(**************************************** WARNING ********************************************
 *** The KEBA Kemro K2 System including software is not intended for safety control tasks! ***
 ***                       For further information see Comment tab!                        ***
 *********************************************************************************************)

IF NOT mbInitDone THEN
    RETURN;
END_IF;

// update lintab
aUpdateLintabOut();

;#END_EDIT_BLOCK END_ALGORITHM

END_ALGORITHM_BLOCK

#END_OF_IEC_PART

@Puma @IecEditor 6 60 @Pou 25
@@@BEG_Comment@@@

@@@END_Comment@@@

@BEG_Contents

@BEG_Func
@RT(17)FuncTreeContainer
0
@END_Func

@BEG_Const
@RT(18)ConstTreeContainer
0
@END_Const

@BEG_Export

@BEG_Kind
@ALGORITHM_BLOCK @RT(24)ABUpdateRelLintabVelCore @STRUCTURED_TEXT
@RT(0) @RT(0) @RT(0)
@END_Kind

@BEG_Dcl
@RT(16)DclTreeContainer
6
@Var @RT(9)PU_Task_7 @RT(0) @T @F @DT @RT(4)TASK @RT(0) @T @T @BASIC 0 @F
@F @F
@T
@BEG_Attrib
3 @RT(0) @RT(0) @RT(0)
@END_Attrib
1 7 @F @F @F @F

@Var @RT(11)mpLintabOut @RT(0) @T @T @REFTO 0 @F @DERIVED 0 @T @T @DT @RT(16)KAPPL_LintabData @RT(0) @T @T @UNKNOWN 0 @F
@F @F
@T
@BEG_Attrib
3 @RT(0) @RT(32)OUT: velocity lintab of movement @RT(0)
@END_Attrib
1 0 @F @F @F @F

@Var @RT(10)mprAbsFlow @RT(0) @T @T @REFTO 0 @T @DT @RT(4)REAL @RT(0) @T @T @BASIC 0 @F
@F @F
@T
@BEG_Attrib
3 @RT(0) @RT(34)IN: maximum absolute flow in l/min @RT(0)
@END_Attrib
1 0 @F @F @F @F

@Var @RT(11)mprMaxSpeed @RT(0) @T @T @REFTO 0 @T @DT @RT(4)REAL @RT(0) @T @T @BASIC 0 @F
@F @F
@T
@BEG_Attrib
3 @RT(0) @RT(33)IN/OUT: max speed of fwd movement @RT(0)
@END_Attrib
1 0 @F @F @F @F

@Var @RT(10)mbInitDone @RT(0) @T @F @DT @RT(4)BOOL @RT(0) @T @T @BASIC 0 @F
@F @F
@T
@BEG_Attrib
3 @RT(0) @RT(0) @RT(0)
@END_Attrib
1 0 @F @F @F @F

@Var @RT(28)sv_bCalcMaxValuesFromCylData @RT(0) @T @F @DT @RT(4)BOOL @RT(0) @T @T @BASIC 0 @F
@F @F
@T
@BEG_Attrib
3 @RT(0) @RT(117)TRUE: calculate max speed and max pressure values by using cylinder data;  FALSE: max values must be entered manually @RT(0)
@END_Attrib
1 8 @F @F @F @F

@END_Dcl

@END_Export

@BEG_Body

5

@BEG_Export

@BEG_Algo
@ALGORITHM @RT(16)aUpdateLintabOut @STRUCTURED_TEXT
@RT(0) @RT(0) @RT(0) @F @F
@END_Algo

@BEG_Dcl
@RT(16)DclTreeContainer
0
@END_Dcl

@END_Export

@BEG_Export

@BEG_Algo
@ALGORITHM @RT(13)aCalcMaxSpeed @STRUCTURED_TEXT
@RT(0) @RT(0) @RT(0) @F @F
@END_Algo

@BEG_Dcl
@RT(16)DclTreeContainer
0
@END_Dcl

@END_Export

@BEG_Export

@BEG_Algo
@ALGORITHM @RT(5)aInit @STRUCTURED_TEXT
@RT(0) @RT(0) @RT(0) @F @F
@END_Algo

@BEG_Dcl
@RT(16)DclTreeContainer
4
@Var @RT(10)pLintabOut @RT(0) @T @T @REFTO 0 @F @DERIVED 0 @T @T @DT @RT(16)KAPPL_LintabData @RT(0) @T @T @UNKNOWN 0 @F
@F @F
@T
@BEG_Attrib
3 @RT(0) @RT(0) @RT(0)
@END_Attrib
1 1 @F @F @F @F

@Var @RT(10)prMaxSpeed @RT(0) @T @T @REFTO 0 @T @DT @RT(4)REAL @RT(0) @T @T @BASIC 0 @F
@F @F
@T
@BEG_Attrib
3 @RT(0) @RT(0) @RT(0)
@END_Attrib
1 1 @F @F @F @F

@Var @RT(9)prAbsFlow @RT(0) @T @T @REFTO 0 @T @DT @RT(4)REAL @RT(0) @T @T @BASIC 0 @F
@F @F
@T
@BEG_Attrib
3 @RT(0) @RT(22)absolute flow in l/min @RT(0)
@END_Attrib
1 1 @F @F @F @F

@Var @RT(3)tmp @RT(0) @T @F @DT @RT(4)DINT @RT(0) @T @T @BASIC 0 @F
@F @F
@T
@BEG_Attrib
3 @RT(0) @RT(0) @RT(0)
@END_Attrib
1 0 @F @F @F @F

@END_Dcl

@END_Export

@BEG_Export

@BEG_Algo
@POSTUPDATE_ALGORITHM @RT(15)pUpdateVelocity @STRUCTURED_TEXT
@RT(0) @RT(11)mprAbsFlow^ @RT(9)PU_Task_7 @F @F
@END_Algo

@BEG_Dcl
@RT(16)DclTreeContainer
0
@END_Dcl

@END_Export

@BEG_Export

@BEG_Algo
@POSTUPDATE_ALGORITHM @RT(21)pUpdateVelocityLintab @STRUCTURED_TEXT
@RT(0) @RT(12)mprMaxSpeed^ @RT(9)PU_Task_7 @F @F
@END_Algo

@BEG_Dcl
@RT(16)DclTreeContainer
0
@END_Dcl

@END_Export

@BEG_Body
@TL(12)
(**************************************** WARNING ********************************************
 *** The KEBA Kemro K2 System including software is not intended for safety control tasks! ***
 ***                       For further information see Comment tab!                        ***
 *********************************************************************************************)

// save data to Vel lintab
mpLintabOut^.LintabPoints.uNoOfPoints := 2;
mpLintabOut^.LintabPoints.Point[1].rX := 0.0;
mpLintabOut^.LintabPoints.Point[1].rY := 0.0;
mpLintabOut^.LintabPoints.Point[2].rX := mprMaxSpeed^;
mpLintabOut^.LintabPoints.Point[2].rY := 100.0; // %

@END_Body

@@@BEG_Comment@@@
@TL(0)

@@@END_Comment@@@

@BEG_Body
@TL(13)
(**************************************** WARNING ********************************************
 *** The KEBA Kemro K2 System including software is not intended for safety control tasks! ***
 ***                       For further information see Comment tab!                        ***
 *********************************************************************************************)

IF NOT sv_bCalcMaxValuesFromCylData THEN
   // no calculation necessary
   RETURN;
END_IF;

// max flow in l/min
mprMaxSpeed^ := mprAbsFlow^;

@END_Body

@@@BEG_Comment@@@
@TL(0)

@@@END_Comment@@@

@BEG_Body
@TL(32)
(**************************************** WARNING ********************************************
 *** The KEBA Kemro K2 System including software is not intended for safety control tasks! ***
 ***                       For further information see Comment tab!                        ***
 *********************************************************************************************)

mbInitDone := FALSE;
mprAbsFlow := prAbsFlow;
mpLintabOut := pLintabOut;
mprMaxSpeed := prMaxSpeed;

IF NOT CHECK_REF(prAbsFlow^) THEN
    tmp := Print('prAbsFlow not valid');
    RETURN;
END_IF;

IF (NOT CHECK_REF(pLintabOut^)) THEN
    tmp := Print('pLintabOut not valid');
    RETURN;
END_IF;

IF (NOT CHECK_REF(prMaxSpeed^)) THEN
    tmp := Print('prMaxSpeed not valid');
    RETURN;
END_IF;

// init successful
mbInitDone := TRUE;

aCalcMaxSpeed();

aUpdateLintabOut();

@END_Body

@@@BEG_Comment@@@
@TL(0)

@@@END_Comment@@@

@BEG_Body
@TL(15)
(**************************************** WARNING ********************************************
 *** The KEBA Kemro K2 System including software is not intended for safety control tasks! ***
 ***                       For further information see Comment tab!                        ***
 *********************************************************************************************)

IF NOT mbInitDone THEN
    RETURN;
END_IF;

aCalcMaxSpeed();

@END_Body

@@@BEG_Comment@@@
@TL(0)

@@@END_Comment@@@

@BEG_Body
@TL(14)
(**************************************** WARNING ********************************************
 *** The KEBA Kemro K2 System including software is not intended for safety control tasks! ***
 ***                       For further information see Comment tab!                        ***
 *********************************************************************************************)

IF NOT mbInitDone THEN
    RETURN;
END_IF;

// update lintab
aUpdateLintabOut();

@END_Body

@@@BEG_Comment@@@
@TL(0)

@@@END_Comment@@@
@END_Body

@END_Contents

(* ---- ABUpdateRelLintabVelInject.pu ---- *)
IMPORT_OVER_LISTFILE
 FFixCylinderData
, FCalculateCylinderSize
, FCalcScrewSize
, FScaleAndFloor
, tnDataState
, tsCylinderData

END_IMPORT

ALGORITHM_BLOCK ABUpdateRelLintabVelInject #DUMMY_EDIT_BLOCK

SYSTEM_VAR
 sv_bCalcMaxValuesFromCylData : BOOL (* TRUE: calculate max speed and max pressure values by using cylinder data;  FALSE: max values must be entered manually *);
 sv_DataState : tnDataState;
 sv_iReadMachineDataCount : UDINT;
END_VAR

SYSTEM_OBJECT
 PU_Task_7 : TASK;
 PU_Task_3 : TASK;
END_OBJECT

VAR
 mprAbsFlow : REFTO REAL;
 mpCylinderData : REFTO tsCylinderData;
 mprMaxSpeed : REFTO REAL;
 mprMaxSpeedCalc : REFTO REAL;
 mprMaxSpeedCalib : REFTO REAL (* IN/OUT: max speed of movement (calculated) *);
 mbprMaxSpeedCalibLinked : BOOL := FALSE (* IN/OUT: max speed of movement (calculated) *);
 mprMaxSpeedReducePercent : REFTO REAL (* IN: percentage to reduce max speed *);
 miMaxSpeedDigitsToFloor : SINT := 0 (* IN: max speed digits to floor *);
 mbInitDone : BOOL;
END_VAR

ALGORITHM aCalcMaxVelocity

VAR_TEMP
 tmp : BOOL;
END_VAR

VAR
 rMaxFlow : REAL (* maximum flow in mm^3/sec *);
 rSize : REAL;
 rScalePercent : REAL;
END_VAR
#BEGIN_EDIT_BLOCK
(**************************************** WARNING ********************************************
 *** The KEBA Kemro K2 System including software is not intended for safety control tasks! ***
 ***                       For further information see Comment tab!                        ***
 *********************************************************************************************)

IF NOT sv_bCalcMaxValuesFromCylData THEN
   // no calculation necessary
   RETURN;
END_IF;

// sanity check
tmp := FFixCylinderData(mpCylinderData);

// convert from l/min to mm^3/sec
rMaxFlow := mprAbsFlow^ * 100.0 *100.0 *100.0 / 60.0;

rSize := FCalculateCylinderSize(CylinderData := mpCylinderData^, bSmallSize := mpCylinderData^.bUseSmallSize, bCalcHighPressSize := FALSE);

//speed in mm/s
mprMaxSpeedCalc^ := (rMaxFlow / rSize);
IF ((mbInitDone AND sv_DataState = nReady) AND (mprMaxSpeed^ > mprMaxSpeedCalc^)) THEN
   // prevent recalculation on machine data load except if max. value exceeds custom value
   rScalePercent := 100.0;
   IF mprMaxSpeedReducePercent <> EMPTY THEN
      rScalePercent := 100.0 - mprMaxSpeedReducePercent^;
   END_IF;
   mprMaxSpeed^ := FScaleAndFloor(mprMaxSpeedCalc^, rScalePercent, miMaxSpeedDigitsToFloor);
END_IF;
// check max velocity for visualization
IF (mbprMaxSpeedCalibLinked) THEN
   IF(mprMaxSpeedCalib^ <= 0.0) OR (mprMaxSpeedCalib^ > mprMaxSpeedCalc^) THEN
      mprMaxSpeedCalib^ := mprMaxSpeedCalc^;
   END_IF;
END_IF;

;#END_EDIT_BLOCK END_ALGORITHM

ALGORITHM aInit

VAR_INPUT
 prMaxSpeed : REFTO REAL (* IN/OUT: max speed of movement *);
 prMaxSpeedCalc : REFTO REAL (* IN/OUT: max speed  calculated of movement *);
 prAbsFlow : REFTO REAL (* IN: maximum absolute flow in l/min *);
 prMaxSpeedReducePercent : REFTO REAL (* IN: reduce max. speed percentage *);
 pCylinderData : REFTO tsCylinderData (* IN: cylinder data *);
 iMaxSpeedDigitsToFloor : SINT;
 prMaxSpeedCalib : REFTO REAL;
END_VAR

VAR
 tmp : DINT;
END_VAR
#BEGIN_EDIT_BLOCK
(**************************************** WARNING ********************************************
 *** The KEBA Kemro K2 System including software is not intended for safety control tasks! ***
 ***                       For further information see Comment tab!                        ***
 *********************************************************************************************)

mbInitDone := FALSE;
mprAbsFlow := prAbsFlow;
mpCylinderData := pCylinderData;
mprMaxSpeed := prMaxSpeed;
mprMaxSpeedCalc := prMaxSpeedCalc;
mprMaxSpeedCalib := prMaxSpeedCalib;
mprMaxSpeedReducePercent := prMaxSpeedReducePercent;
miMaxSpeedDigitsToFloor := iMaxSpeedDigitsToFloor;

IF NOT CHECK_REF(prAbsFlow^) THEN
    tmp := Print('prAbsFlow not valid');
    RETURN;
END_IF;

IF NOT CHECK_REF(pCylinderData^) THEN
    tmp := Print('pCylinderData not valid');
    RETURN;
END_IF;

IF NOT CHECK_REF(prMaxSpeed^) THEN
    tmp := Print('at least one prMaxSpeedxxx not valid');
    RETURN;
END_IF;

IF NOT CHECK_REF(prMaxSpeedCalc^) THEN
    tmp := Print('prMaxSpeedCalc not valid');
    RETURN;
END_IF;

IF (CHECK_REF(mprMaxSpeedCalib^)) THEN
    mbprMaxSpeedCalibLinked := TRUE;
END_IF;

// calculate
aCalcMaxVelocity();

// init successful
mbInitDone := TRUE;

;#END_EDIT_BLOCK END_ALGORITHM

POSTUPDATE_ALGORITHM pUpdateVelocity ON PU_Task_7 WITH mprAbsFlow^,mpCylinderData^

#BEGIN_EDIT_BLOCK
(**************************************** WARNING ********************************************
 *** The KEBA Kemro K2 System including software is not intended for safety control tasks! ***
 ***                       For further information see Comment tab!                        ***
 *********************************************************************************************)

IF NOT mbInitDone OR (sv_DataState = nReadMachineData) THEN
   RETURN;
END_IF;

// reset calib value if diameter or flow is changed
IF (mbprMaxSpeedCalibLinked AND (sv_DataState = nReady)) THEN
   mprMaxSpeedCalib^ := 0.0;
END_IF;

aCalcMaxVelocity();

;#END_EDIT_BLOCK END_ALGORITHM

POSTUPDATE_ALGORITHM pUpdateMaxVelocity ON PU_Task_7 WITH mprMaxSpeedCalib^

VAR
 rScalePercent : REAL;
END_VAR
#BEGIN_EDIT_BLOCK
(**************************************** WARNING ********************************************
 *** The KEBA Kemro K2 System including software is not intended for safety control tasks! ***
 ***                       For further information see Comment tab!                        ***
 *********************************************************************************************)

IF sv_DataState = nReadMachineData THEN
   RETURN;
END_IF;

IF ((mprMaxSpeedCalib^ < mprMaxSpeed^) AND (mprMaxSpeedCalib^ > 0.0)) THEN
   rScalePercent := 100.0;
   IF mprMaxSpeedReducePercent <> EMPTY THEN
      rScalePercent := 100.0 - mprMaxSpeedReducePercent^;
   END_IF;
   mprMaxSpeed^ := FScaleAndFloor(mprMaxSpeedCalib^, rScalePercent, miMaxSpeedDigitsToFloor);
END_IF;

;#END_EDIT_BLOCK END_ALGORITHM

POSTUPDATE_ALGORITHM pMachineDataLoaded ON PU_Task_7 WITH sv_iReadMachineDataCount

#BEGIN_EDIT_BLOCK
(**************************************** WARNING ********************************************
 *** The KEBA Kemro K2 System including software is not intended for safety control tasks! ***
 ***                       For further information see Comment tab!                        ***
 *********************************************************************************************)

aCalcMaxVelocity();

;#END_EDIT_BLOCK END_ALGORITHM

POSTUPDATE_ALGORITHM pMachineDataLoadingStarted ON PU_Task_3(1) WITH sv_DataState

#BEGIN_EDIT_BLOCK
(**************************************** WARNING ********************************************
 *** The KEBA Kemro K2 System including software is not intended for safety control tasks! ***
 ***                       For further information see Comment tab!                        ***
 *********************************************************************************************)

IF sv_DataState = nReadMachineData THEN
   //reset max speed calib at the beginning of machine data loading
   //if max speed calib is part of the loaded machine data, the correct value comes from the XMl file
   //if max speed calib is not part of machine data it is set to max speed calc
   //when calling aCalcMaxVelocity after loading machine data is finished
   IF mbprMaxSpeedCalibLinked THEN
      mprMaxSpeedCalib^ := 0.0;
   END_IF;
END_IF;

;#END_EDIT_BLOCK END_ALGORITHM

END_ALGORITHM_BLOCK

#END_OF_IEC_PART

@Puma @IecEditor 6 114 @Pou 25
@@@BEG_Comment@@@

@@@END_Comment@@@

@BEG_Contents

@BEG_Func
@RT(17)FuncTreeContainer
4
@Var @RT(16)FFixCylinderData @RT(0) @T @T @DERIVED 0 @F @RT(8)FUNCTION @F
@T
@BEG_Attrib
0 @RT(0) @RT(0)
@END_Attrib
1 1 @F @F @F @F

@Var @RT(22)FCalculateCylinderSize @RT(0) @T @T @DERIVED 0 @F @RT(8)FUNCTION @F
@T
@BEG_Attrib
0 @RT(0) @RT(0)
@END_Attrib
1 1 @F @F @F @F

@Var @RT(14)FCalcScrewSize @RT(0) @T @T @DERIVED 0 @F @RT(8)FUNCTION @F
@T
@BEG_Attrib
0 @RT(0) @RT(0)
@END_Attrib
1 1 @F @F @F @F

@Var @RT(14)FScaleAndFloor @RT(0) @T @T @DERIVED 0 @F @RT(8)FUNCTION @F
@T
@BEG_Attrib
0 @RT(0) @RT(0)
@END_Attrib
1 1 @F @F @F @F

@END_Func

@BEG_Const
@RT(18)ConstTreeContainer
0
@END_Const

@BEG_Export

@BEG_Kind
@ALGORITHM_BLOCK @RT(26)ABUpdateRelLintabVelInject @STRUCTURED_TEXT
@RT(0) @RT(0) @RT(0)
@END_Kind

@BEG_Dcl
@RT(16)DclTreeContainer
14
@Var @RT(28)sv_bCalcMaxValuesFromCylData @RT(0) @T @F @DT @RT(4)BOOL @RT(0) @T @T @BASIC 0 @F
@F @F
@T
@BEG_Attrib
3 @RT(0) @RT(117)TRUE: calculate max speed and max pressure values by using cylinder data;  FALSE: max values must be entered manually @RT(0)
@END_Attrib
1 8 @F @F @F @F

@Var @RT(12)sv_DataState @RT(0) @T @T @DERIVED 0 @T @T @DT @RT(11)tnDataState @RT(0) @T @T @UNKNOWN 0 @F
@F @F
@T
@BEG_Attrib
3 @RT(0) @RT(0) @RT(0)
@END_Attrib
1 8 @F @F @F @F

@Var @RT(9)PU_Task_7 @RT(0) @T @F @DT @RT(4)TASK @RT(0) @T @T @BASIC 0 @F
@F @F
@T
@BEG_Attrib
3 @RT(0) @RT(0) @RT(0)
@END_Attrib
1 7 @F @F @F @F

@Var @RT(10)mprAbsFlow @RT(0) @T @T @REFTO 0 @T @DT @RT(4)REAL @RT(0) @T @T @BASIC 0 @F
@F @F
@T
@BEG_Attrib
3 @RT(0) @RT(0) @RT(0)
@END_Attrib
1 0 @F @F @F @F

@Var @RT(14)mpCylinderData @RT(0) @T @T @REFTO 0 @F @DERIVED 0 @T @T @DT @RT(14)tsCylinderData @RT(0) @T @T @UNKNOWN 0 @F
@F @F
@T
@BEG_Attrib
3 @RT(0) @RT(0) @RT(0)
@END_Attrib
1 0 @F @F @F @F

@Var @RT(11)mprMaxSpeed @RT(0) @T @T @REFTO 0 @T @DT @RT(4)REAL @RT(0) @T @T @BASIC 0 @F
@F @F
@T
@BEG_Attrib
3 @RT(0) @RT(0) @RT(0)
@END_Attrib
1 0 @F @F @F @F

@Var @RT(15)mprMaxSpeedCalc @RT(0) @T @T @REFTO 0 @T @DT @RT(4)REAL @RT(0) @T @T @BASIC 0 @F
@F @F
@T
@BEG_Attrib
3 @RT(0) @RT(0) @RT(0)
@END_Attrib
1 0 @F @F @F @F

@Var @RT(16)mprMaxSpeedCalib @RT(0) @T @T @REFTO 0 @T @DT @RT(4)REAL @RT(0) @T @T @BASIC 0 @F
@F @F
@T
@BEG_Attrib
3 @RT(0) @RT(42)IN/OUT: max speed of movement (calculated) @RT(0)
@END_Attrib
1 0 @F @F @F @F

@Var @RT(23)mbprMaxSpeedCalibLinked @RT(0) @T @F @DT @RT(4)BOOL @RT(0) @T @T @BASIC 0 @F
@F @F
@T
@BEG_Attrib
3 @RT(5)FALSE @RT(42)IN/OUT: max speed of movement (calculated) @RT(0)
@END_Attrib
1 0 @F @F @F @F

@Var @RT(24)mprMaxSpeedReducePercent @RT(0) @T @T @REFTO 0 @T @DT @RT(4)REAL @RT(0) @T @T @BASIC 0 @F
@F @F
@T
@BEG_Attrib
3 @RT(0) @RT(34)IN: percentage to reduce max speed @RT(0)
@END_Attrib
1 0 @F @F @F @F

@Var @RT(23)miMaxSpeedDigitsToFloor @RT(0) @T @F @DT @RT(4)SINT @RT(0) @T @T @BASIC 0 @F
@F @F
@T
@BEG_Attrib
3 @RT(1)0 @RT(29)IN: max speed digits to floor @RT(0)
@END_Attrib
1 0 @F @F @F @F

@Var @RT(10)mbInitDone @RT(0) @T @F @DT @RT(4)BOOL @RT(0) @T @T @BASIC 0 @F
@F @F
@T
@BEG_Attrib
3 @RT(0) @RT(0) @RT(0)
@END_Attrib
1 0 @F @F @F @F

@Var @RT(24)sv_iReadMachineDataCount @RT(0) @T @T @RENAMED 0 @T @T @DT @RT(5)UDINT @RT(0) @T @T @BASIC 0 @F
@F @F
@T
@BEG_Attrib
3 @RT(0) @RT(0) @RT(0)
@END_Attrib
1 8 @F @F @F @F

@Var @RT(9)PU_Task_3 @RT(0) @T @T @RENAMED 0 @T @T @DT @RT(4)TASK @RT(0) @T @T @BASIC 0 @F
@F @F
@T
@BEG_Attrib
3 @RT(0) @RT(0) @RT(0)
@END_Attrib
1 7 @F @F @F @F

@END_Dcl

@END_Export

@BEG_Body

6

@BEG_Export

@BEG_Algo
@ALGORITHM @RT(16)aCalcMaxVelocity @STRUCTURED_TEXT
@RT(0) @RT(0) @RT(0) @F @F
@END_Algo

@BEG_Dcl
@RT(16)DclTreeContainer
4
@Var @RT(3)tmp @RT(0) @T @F @DT @RT(4)BOOL @RT(0) @T @T @BASIC 0 @F
@F @F
@T
@BEG_Attrib
3 @RT(0) @RT(0) @RT(0)
@END_Attrib
1 4 @F @F @F @F

@Var @RT(8)rMaxFlow @RT(0) @T @F @DT @RT(4)REAL @RT(0) @T @T @BASIC 0 @F
@F @F
@T
@BEG_Attrib
3 @RT(0) @RT(24)maximum flow in mm^3/sec @RT(0)
@END_Attrib
1 0 @F @F @F @F

@Var @RT(5)rSize @RT(0) @T @F @DT @RT(4)REAL @RT(0) @T @T @BASIC 0 @F
@F @F
@T
@BEG_Attrib
3 @RT(0) @RT(0) @RT(0)
@END_Attrib
1 0 @F @F @F @F

@Var @RT(13)rScalePercent @RT(0) @T @F @DT @RT(4)REAL @RT(0) @T @T @BASIC 0 @F
@F @F
@T
@BEG_Attrib
3 @RT(0) @RT(0) @RT(0)
@END_Attrib
1 0 @F @F @F @F

@END_Dcl

@END_Export

@BEG_Export

@BEG_Algo
@ALGORITHM @RT(5)aInit @STRUCTURED_TEXT
@RT(0) @RT(0) @RT(0) @F @F
@END_Algo

@BEG_Dcl
@RT(16)DclTreeContainer
8
@Var @RT(10)prMaxSpeed @RT(0) @T @T @REFTO 0 @T @DT @RT(4)REAL @RT(0) @T @T @BASIC 0 @F
@F @F
@T
@BEG_Attrib
3 @RT(0) @RT(29)IN/OUT: max speed of movement @RT(0)
@END_Attrib
1 1 @F @F @F @F

@Var @RT(14)prMaxSpeedCalc @RT(0) @T @T @REFTO 0 @T @DT @RT(4)REAL @RT(0) @T @T @BASIC 0 @F
@F @F
@T
@BEG_Attrib
3 @RT(0) @RT(41)IN/OUT: max speed  calculated of movement @RT(0)
@END_Attrib
1 1 @F @F @F @F

@Var @RT(9)prAbsFlow @RT(0) @T @T @REFTO 0 @T @DT @RT(4)REAL @RT(0) @T @T @BASIC 0 @F
@F @F
@T
@BEG_Attrib
3 @RT(0) @RT(34)IN: maximum absolute flow in l/min @RT(0)
@END_Attrib
1 1 @F @F @F @F

@Var @RT(23)prMaxSpeedReducePercent @RT(0) @T @T @REFTO 0 @T @DT @RT(4)REAL @RT(0) @T @T @BASIC 0 @F
@F @F
@T
@BEG_Attrib
3 @RT(0) @RT(32)IN: reduce max. speed percentage @RT(0)
@END_Attrib
1 1 @F @F @F @F

@Var @RT(13)pCylinderData @RT(0) @T @T @REFTO 0 @F @DERIVED 0 @T @T @DT @RT(14)tsCylinderData @RT(0) @T @T @UNKNOWN 0 @F
@F @F
@T
@BEG_Attrib
3 @RT(0) @RT(17)IN: cylinder data @RT(0)
@END_Attrib
1 1 @F @F @F @F

@Var @RT(3)tmp @RT(0) @T @F @DT @RT(4)DINT @RT(0) @T @T @BASIC 0 @F
@F @F
@T
@BEG_Attrib
3 @RT(0) @RT(0) @RT(0)
@END_Attrib
1 0 @F @F @F @F

@Var @RT(22)iMaxSpeedDigitsToFloor @RT(0) @T @F @DT @RT(4)SINT @RT(0) @T @T @BASIC 0 @F
@F @F
@T
@BEG_Attrib
3 @RT(0) @RT(0) @RT(0)
@END_Attrib
1 1 @F @F @F @F

@Var @RT(15)prMaxSpeedCalib @RT(0) @T @T @REFTO 0 @T @DT @RT(4)REAL @RT(0) @T @T @BASIC 0 @F
@F @F
@T
@BEG_Attrib
3 @RT(0) @RT(0) @RT(0)
@END_Attrib
1 1 @F @F @F @F

@END_Dcl

@END_Export

@BEG_Export

@BEG_Algo
@POSTUPDATE_ALGORITHM @RT(15)pUpdateVelocity @STRUCTURED_TEXT
@RT(0) @RT(27)mprAbsFlow^,mpCylinderData^ @RT(9)PU_Task_7 @F @F
@END_Algo

@BEG_Dcl
@RT(16)DclTreeContainer
0
@END_Dcl

@END_Export

@BEG_Export

@BEG_Algo
@POSTUPDATE_ALGORITHM @RT(18)pUpdateMaxVelocity @STRUCTURED_TEXT
@RT(0) @RT(17)mprMaxSpeedCalib^ @RT(9)PU_Task_7 @F @F
@END_Algo

@BEG_Dcl
@RT(16)DclTreeContainer
1
@Var @RT(13)rScalePercent @RT(0) @T @F @DT @RT(4)REAL @RT(0) @T @T @BASIC 0 @F
@F @F
@T
@BEG_Attrib
3 @RT(0) @RT(0) @RT(0)
@END_Attrib
1 0 @F @F @F @F

@END_Dcl

@END_Export

@BEG_Export

@BEG_Algo
@POSTUPDATE_ALGORITHM @RT(18)pMachineDataLoaded @STRUCTURED_TEXT
@RT(0) @RT(24)sv_iReadMachineDataCount @RT(9)PU_Task_7 @F @F
@END_Algo

@BEG_Dcl
@RT(16)DclTreeContainer
0
@END_Dcl

@END_Export

@BEG_Export

@BEG_Algo
@POSTUPDATE_ALGORITHM @RT(26)pMachineDataLoadingStarted @STRUCTURED_TEXT
@RT(0) @RT(12)sv_DataState @RT(12)PU_Task_3(1) @F @F
@END_Algo

@BEG_Dcl
@RT(16)DclTreeContainer
0
@END_Dcl

@END_Export

@BEG_Body
@TL(35)
(**************************************** WARNING ********************************************
 *** The KEBA Kemro K2 System including software is not intended for safety control tasks! ***
 ***                       For further information see Comment tab!                        ***
 *********************************************************************************************)

IF NOT sv_bCalcMaxValuesFromCylData THEN
   // no calculation necessary
   RETURN;
END_IF;

// sanity check
tmp := FFixCylinderData(mpCylinderData);

// convert from l/min to mm^3/sec
rMaxFlow := mprAbsFlow^ * 100.0 *100.0 *100.0 / 60.0;

rSize := FCalculateCylinderSize(CylinderData := mpCylinderData^, bSmallSize := mpCylinderData^.bUseSmallSize, bCalcHighPressSize := FALSE);

//speed in mm/s
mprMaxSpeedCalc^ := (rMaxFlow / rSize);
IF ((mbInitDone AND sv_DataState = nReady) AND (mprMaxSpeed^ > mprMaxSpeedCalc^)) THEN
   // prevent recalculation on machine data load except if max. value exceeds custom value
   rScalePercent := 100.0;
   IF mprMaxSpeedReducePercent <> EMPTY THEN
      rScalePercent := 100.0 - mprMaxSpeedReducePercent^;
   END_IF;
   mprMaxSpeed^ := FScaleAndFloor(mprMaxSpeedCalc^, rScalePercent, miMaxSpeedDigitsToFloor);
END_IF;
// check max velocity for visualization
IF (mbprMaxSpeedCalibLinked) THEN
   IF(mprMaxSpeedCalib^ <= 0.0) OR (mprMaxSpeedCalib^ > mprMaxSpeedCalc^) THEN
      mprMaxSpeedCalib^ := mprMaxSpeedCalc^;
   END_IF;
END_IF;

@END_Body

@@@BEG_Comment@@@
@TL(0)

@@@END_Comment@@@

@BEG_Body
@TL(46)
(**************************************** WARNING ********************************************
 *** The KEBA Kemro K2 System including software is not intended for safety control tasks! ***
 ***                       For further information see Comment tab!                        ***
 *********************************************************************************************)

mbInitDone := FALSE;
mprAbsFlow := prAbsFlow;
mpCylinderData := pCylinderData;
mprMaxSpeed := prMaxSpeed;
mprMaxSpeedCalc := prMaxSpeedCalc;
mprMaxSpeedCalib := prMaxSpeedCalib;
mprMaxSpeedReducePercent := prMaxSpeedReducePercent;
miMaxSpeedDigitsToFloor := iMaxSpeedDigitsToFloor;

IF NOT CHECK_REF(prAbsFlow^) THEN
    tmp := Print('prAbsFlow not valid');
    RETURN;
END_IF;

IF NOT CHECK_REF(pCylinderData^) THEN
    tmp := Print('pCylinderData not valid');
    RETURN;
END_IF;

IF NOT CHECK_REF(prMaxSpeed^) THEN
    tmp := Print('at least one prMaxSpeedxxx not valid');
    RETURN;
END_IF;

IF NOT CHECK_REF(prMaxSpeedCalc^) THEN
    tmp := Print('prMaxSpeedCalc not valid');
    RETURN;
END_IF;

IF (CHECK_REF(mprMaxSpeedCalib^)) THEN
    mbprMaxSpeedCalibLinked := TRUE;
END_IF;

// calculate
aCalcMaxVelocity();

// init successful
mbInitDone := TRUE;

@END_Body

@@@BEG_Comment@@@
@TL(0)

@@@END_Comment@@@

@BEG_Body
@TL(20)
(**************************************** WARNING ********************************************
 *** The KEBA Kemro K2 System including software is not intended for safety control tasks! ***
 ***                       For further information see Comment tab!                        ***
 *********************************************************************************************)

IF NOT mbInitDone OR (sv_DataState = nReadMachineData) THEN
   RETURN;
END_IF;

// reset calib value if diameter or flow is changed
IF (mbprMaxSpeedCalibLinked AND (sv_DataState = nReady)) THEN
   mprMaxSpeedCalib^ := 0.0;
END_IF;

aCalcMaxVelocity();

@END_Body

@@@BEG_Comment@@@
@TL(0)

@@@END_Comment@@@

@BEG_Body
@TL(18)
(**************************************** WARNING ********************************************
 *** The KEBA Kemro K2 System including software is not intended for safety control tasks! ***
 ***                       For further information see Comment tab!                        ***
 *********************************************************************************************)

IF sv_DataState = nReadMachineData THEN
   RETURN;
END_IF;

IF ((mprMaxSpeedCalib^ < mprMaxSpeed^) AND (mprMaxSpeedCalib^ > 0.0)) THEN
   rScalePercent := 100.0;
   IF mprMaxSpeedReducePercent <> EMPTY THEN
      rScalePercent := 100.0 - mprMaxSpeedReducePercent^;
   END_IF;
   mprMaxSpeed^ := FScaleAndFloor(mprMaxSpeedCalib^, rScalePercent, miMaxSpeedDigitsToFloor);
END_IF;

@END_Body

@@@BEG_Comment@@@
@TL(0)

@@@END_Comment@@@

@BEG_Body
@TL(7)
(**************************************** WARNING ********************************************
 *** The KEBA Kemro K2 System including software is not intended for safety control tasks! ***
 ***                       For further information see Comment tab!                        ***
 *********************************************************************************************)

aCalcMaxVelocity();

@END_Body

@@@BEG_Comment@@@
@TL(0)

@@@END_Comment@@@

@BEG_Body
@TL(15)
(**************************************** WARNING ********************************************
 *** The KEBA Kemro K2 System including software is not intended for safety control tasks! ***
 ***                       For further information see Comment tab!                        ***
 *********************************************************************************************)

IF sv_DataState = nReadMachineData THEN
   //reset max speed calib at the beginning of machine data loading
   //if max speed calib is part of the loaded machine data, the correct value comes from the XMl file
   //if max speed calib is not part of machine data it is set to max speed calc
   //when calling aCalcMaxVelocity after loading machine data is finished
   IF mbprMaxSpeedCalibLinked THEN
      mprMaxSpeedCalib^ := 0.0;
   END_IF;
END_IF;

@END_Body

@@@BEG_Comment@@@
@TL(0)

@@@END_Comment@@@
@END_Body

@END_Contents

(* ---- ABUpdateRelLintabVelPlast.pu ---- *)
(*
@h    ! WARNING !
@h    The Kemro K2 system (including software) only meets category B according to EN 954-1,
@h    thus it is not intended for usage in safety-relevant control applications in the field
@h    of personal safety (e.g. emergency stop).
@h    To implement potentially necessary safety-relevant control tasks, always use additional
@h    external safety devices that are intended for the particular purpose, and meet the necessary
@h    functional safety.
@h    For further information see EN 954-1 (EN ISO 13849-1) and/or the K2-x00 user manual, chapter
@h    "CE conformity, directives and standards".

same as ABUpdateRelLintab, but only updates pressure lintab
also there is only one direction
used for updating RPM lintab
*)

IMPORT_OVER_LISTFILE
 FCalcScrewCircumfenceSpeed
, FScaleAndFloor
, tnDataState
, KAPPL_LintabData

END_IMPORT

ALGORITHM_BLOCK ABUpdateRelLintabVelPlast #DUMMY_EDIT_BLOCK

SYSTEM_VAR
 sv_DataState : tnDataState;
 sv_iReadMachineDataCount : UDINT;
END_VAR

SYSTEM_OBJECT
 PU_Task_7 : TASK;
END_OBJECT

VAR
 mpLintabInV : REFTO KAPPL_LintabData;
 mpLintabOutV : REFTO KAPPL_LintabData;
 mprMaxSpeed : REFTO REAL;
 mbInitDone : BOOL;
 mprScrewDiameter : REFTO REAL;
 mprMaxRPM : REFTO REAL (* max. RPM from calibration *);
 mprMaxRPMProfile : REFTO REAL (* max. RPM used for profiles *);
 mprMaxRPMReducePercent : REFTO REAL (* profile RPM reduce percentage (0-100%) *);
 miMaxRPMDigitsToFloor : SINT := 0 (* significant digits to floor for RPM profile *);
END_VAR

ALGORITHM aUpdateLintabOut

VAR_TEMP
 i : UDINT;
END_VAR
#BEGIN_EDIT_BLOCK
(**************************************** WARNING ********************************************
 *** The KEBA Kemro K2 System including software is not intended for safety control tasks! ***
 ***                       For further information see Comment tab!                        ***
 *********************************************************************************************)

(* convert lintab from RPM to cm/s screw circumfence speed *)
FOR i := 1 TO mpLintabInV^.LintabPoints.uNoOfPoints DO
   mpLintabOutV^.LintabPoints.Point[i].rX := FCalcScrewCircumfenceSpeed(rDiameter := mprScrewDiameter^, rRPM := mpLintabInV^.LintabPoints.Point[i].rX);// * rTmp;
   mpLintabOutV^.LintabPoints.Point[i].rY := mpLintabInV^.LintabPoints.Point[i].rY;
END_FOR;
mpLintabOutV^.LintabPoints.uNoOfPoints := mpLintabInV^.LintabPoints.uNoOfPoints;

;#END_EDIT_BLOCK END_ALGORITHM

ALGORITHM aCalcMaxSpeed

#BEGIN_EDIT_BLOCK
(**************************************** WARNING ********************************************
 *** The KEBA Kemro K2 System including software is not intended for safety control tasks! ***
 ***                       For further information see Comment tab!                        ***
 *********************************************************************************************)

mprMaxSpeed^ := FCalcScrewCircumfenceSpeed(rDiameter := mprScrewDiameter^, rRPM := mprMaxRPMProfile^);

;#END_EDIT_BLOCK END_ALGORITHM

(*
update pressure / speed lintabs for plast movement

update pLintabOutP and pLintabOutV according to the other parameters
the out lintab is updated when one of the input parameters changes
prMaxPressure points to the max pressure variable of the movement
prMaxSpeed is the maximum circumfence speed of the screw
it will be updated when max RPM input value or the prScrewDiameter changes
*)

ALGORITHM aInit

VAR_INPUT
 prScrewDiameter : REFTO REAL (* IN: screw diameter *);
 prMaxRPM : REFTO REAL (* IN: max RPM of screw *);
 prMaxRPMProfile : REFTO REAL (* IN: max RPM used for profile *);
 prMaxRPMReducePercent : REFTO REAL (* IN: max RPM reduce percentage *);
 iMaxRPMDigitsToFloor : SINT (* IN: max. significant digits to floor for RPM profile *);
 pLintabInV : REFTO KAPPL_LintabData (* IN: screw lintab RPM to % *);
 pLintabOutV : REFTO KAPPL_LintabData (* OUT: screw lintab cm/s to % *);
 prMaxSpeed : REFTO REAL (* OUT: max circumfence speed of screw in cm/s *);
END_VAR

VAR_TEMP
 tmp : DINT;
END_VAR
#BEGIN_EDIT_BLOCK
(**************************************** WARNING ********************************************
 *** The KEBA Kemro K2 System including software is not intended for safety control tasks! ***
 ***                       For further information see Comment tab!                        ***
 *********************************************************************************************)

mbInitDone := FALSE;

IF (NOT CHECK_REF(pLintabInV^)) OR (NOT CHECK_REF(pLintabOutV^)) THEN
    tmp := Print('pLintabInP or pLintabInV not valid');
    RETURN;
END_IF;

IF NOT CHECK_REF(prScrewDiameter^) THEN
    tmp := Print('prMaxPressure not valid');
    RETURN;
END_IF;

IF NOT CHECK_REF(prMaxRPM^) THEN
    tmp := Print('prMaxRPM not valid');
    RETURN;
END_IF;

IF NOT CHECK_REF(prMaxRPMProfile^) THEN
    tmp := Print('prMaxRPMProfile not valid');
    RETURN;
END_IF;

IF NOT CHECK_REF(prMaxRPMReducePercent^) THEN
    tmp := Print('prMaxRPMReducePercent not valid');
    RETURN;
END_IF;

IF NOT CHECK_REF(prMaxSpeed^) THEN
    tmp := Print('prMaxSpeed not valid');
    RETURN;
END_IF;

IF NOT CHECK_REF(prScrewDiameter^) THEN
    tmp := Print('prScrewDiameter not valid');
    RETURN;
END_IF;

mpLintabInV := pLintabInV;
mpLintabOutV := pLintabOutV;
mprScrewDiameter := prScrewDiameter;
mprMaxRPM := prMaxRPM;
mprMaxRPMProfile := prMaxRPMProfile;
mprMaxSpeed := prMaxSpeed;
mprMaxRPMReducePercent := prMaxRPMReducePercent;
miMaxRPMDigitsToFloor := iMaxRPMDigitsToFloor;

// init successful
mbInitDone := TRUE;

aCalcMaxSpeed();

aUpdateLintabOut();

;#END_EDIT_BLOCK END_ALGORITHM

POSTUPDATE_ALGORITHM pUpdateRPM ON PU_Task_7 WITH mprMaxRPM^

VAR
 rScalePercent : REAL := 100.0;
END_VAR
#BEGIN_EDIT_BLOCK
(**************************************** WARNING ********************************************
 *** The KEBA Kemro K2 System including software is not intended for safety control tasks! ***
 ***                       For further information see Comment tab!                        ***
 *********************************************************************************************)

IF NOT mbInitDone OR (sv_DataState = nReadMachineData) THEN
   RETURN;
END_IF;

IF (sv_DataState = nReady AND (mprMaxRPMProfile^ > mprMaxRPM^)) THEN
   // prevent recalculation on machine data load except if max. value exceeds custom value
   IF mprMaxRPMReducePercent <> EMPTY THEN
      rScalePercent := 100.0 - mprMaxRPMReducePercent^;
   END_IF;
   mprMaxRPMProfile^ := FScaleAndFloor(mprMaxRPM^, rScalePercent, miMaxRPMDigitsToFloor);
END_IF;

;#END_EDIT_BLOCK END_ALGORITHM

POSTUPDATE_ALGORITHM pUpdateVelocity ON PU_Task_7 WITH mprScrewDiameter^,mprMaxRPMProfile^

#BEGIN_EDIT_BLOCK
(**************************************** WARNING ********************************************
 *** The KEBA Kemro K2 System including software is not intended for safety control tasks! ***
 ***                       For further information see Comment tab!                        ***
 *********************************************************************************************)

IF NOT mbInitDone OR (sv_DataState = nReadMachineData) THEN
   RETURN;
END_IF;

aCalcMaxSpeed();

;#END_EDIT_BLOCK END_ALGORITHM

POSTUPDATE_ALGORITHM pUpdateVelocityLintab ON PU_Task_7 WITH mprMaxSpeed^,mpLintabInV^

#BEGIN_EDIT_BLOCK
(**************************************** WARNING ********************************************
 *** The KEBA Kemro K2 System including software is not intended for safety control tasks! ***
 ***                       For further information see Comment tab!                        ***
 *********************************************************************************************)

IF NOT mbInitDone THEN
    RETURN;
END_IF;

//update lintab
aUpdateLintabOut();

;#END_EDIT_BLOCK END_ALGORITHM

POSTUPDATE_ALGORITHM pMachineDataLoaded ON PU_Task_7 WITH sv_iReadMachineDataCount

#BEGIN_EDIT_BLOCK
(**************************************** WARNING ********************************************
 *** The KEBA Kemro K2 System including software is not intended for safety control tasks! ***
 ***                       For further information see Comment tab!                        ***
 *********************************************************************************************)

aCalcMaxSpeed();

;#END_EDIT_BLOCK END_ALGORITHM

END_ALGORITHM_BLOCK

#END_OF_IEC_PART

@Puma @IecEditor 6 60 @Pou 25
@@@BEG_Comment@@@
@h    ! WARNING !
@h    The Kemro K2 system (including software) only meets category B according to EN 954-1,
@h    thus it is not intended for usage in safety-relevant control applications in the field
@h    of personal safety (e.g. emergency stop).
@h    To implement potentially necessary safety-relevant control tasks, always use additional
@h    external safety devices that are intended for the particular purpose, and meet the necessary
@h    functional safety.
@h    For further information see EN 954-1 (EN ISO 13849-1) and/or the K2-x00 user manual, chapter
@h    "CE conformity, directives and standards".

same as ABUpdateRelLintab, but only updates pressure lintab
also there is only one direction
used for updating RPM lintab
@@@END_Comment@@@

@BEG_Contents

@BEG_Func
@RT(17)FuncTreeContainer
2
@Var @RT(26)FCalcScrewCircumfenceSpeed @RT(0) @T @T @DERIVED 0 @F @RT(8)FUNCTION @F
@T
@BEG_Attrib
0 @RT(0) @RT(0)
@END_Attrib
1 1 @F @F @F @F

@Var @RT(14)FScaleAndFloor @RT(0) @T @T @DERIVED 0 @F @RT(8)FUNCTION @F
@T
@BEG_Attrib
0 @RT(0) @RT(0)
@END_Attrib
1 1 @F @F @F @F

@END_Func

@BEG_Const
@RT(18)ConstTreeContainer
0
@END_Const

@BEG_Export

@BEG_Kind
@ALGORITHM_BLOCK @RT(25)ABUpdateRelLintabVelPlast @STRUCTURED_TEXT
@RT(0) @RT(0) @RT(0)
@END_Kind

@BEG_Dcl
@RT(16)DclTreeContainer
12
@Var @RT(9)PU_Task_7 @RT(0) @T @F @DT @RT(4)TASK @RT(0) @T @T @BASIC 0 @F
@F @F
@T
@BEG_Attrib
3 @RT(0) @RT(0) @RT(0)
@END_Attrib
1 7 @F @F @F @F

@Var @RT(12)sv_DataState @RT(0) @T @T @DERIVED 0 @T @T @DT @RT(11)tnDataState @RT(0) @T @T @UNKNOWN 0 @F
@F @F
@T
@BEG_Attrib
3 @RT(0) @RT(0) @RT(0)
@END_Attrib
1 8 @F @F @F @F

@Var @RT(11)mpLintabInV @RT(0) @T @T @REFTO 0 @F @DERIVED 0 @T @T @DT @RT(16)KAPPL_LintabData @RT(0) @T @T @UNKNOWN 0 @F
@F @F
@T
@BEG_Attrib
3 @RT(0) @RT(0) @RT(0)
@END_Attrib
1 0 @F @F @F @F

@Var @RT(12)mpLintabOutV @RT(0) @T @T @REFTO 0 @F @DERIVED 0 @T @T @DT @RT(16)KAPPL_LintabData @RT(0) @T @T @UNKNOWN 0 @F
@F @F
@T
@BEG_Attrib
3 @RT(0) @RT(0) @RT(0)
@END_Attrib
1 0 @F @F @F @F

@Var @RT(11)mprMaxSpeed @RT(0) @T @T @REFTO 0 @T @DT @RT(4)REAL @RT(0) @T @T @BASIC 0 @F
@F @F
@T
@BEG_Attrib
3 @RT(0) @RT(0) @RT(0)
@END_Attrib
1 0 @F @F @F @F

@Var @RT(10)mbInitDone @RT(0) @T @F @DT @RT(4)BOOL @RT(0) @T @T @BASIC 0 @F
@F @F
@T
@BEG_Attrib
3 @RT(0) @RT(0) @RT(0)
@END_Attrib
1 0 @F @F @F @F

@Var @RT(16)mprScrewDiameter @RT(0) @T @T @REFTO 0 @T @DT @RT(4)REAL @RT(0) @T @T @BASIC 0 @F
@F @F
@T
@BEG_Attrib
3 @RT(0) @RT(0) @RT(0)
@END_Attrib
1 0 @F @F @F @F

@Var @RT(9)mprMaxRPM @RT(0) @T @T @REFTO 0 @T @DT @RT(4)REAL @RT(0) @T @T @BASIC 0 @F
@F @F
@T
@BEG_Attrib
3 @RT(0) @RT(25)max. RPM from calibration @RT(0)
@END_Attrib
1 0 @F @F @F @F

@Var @RT(16)mprMaxRPMProfile @RT(0) @T @T @REFTO 0 @T @DT @RT(4)REAL @RT(0) @T @T @BASIC 0 @F
@F @F
@T
@BEG_Attrib
3 @RT(0) @RT(26)max. RPM used for profiles @RT(0)
@END_Attrib
1 0 @F @F @F @F

@Var @RT(22)mprMaxRPMReducePercent @RT(0) @T @T @REFTO 0 @T @DT @RT(4)REAL @RT(0) @T @T @BASIC 0 @F
@F @F
@T
@BEG_Attrib
3 @RT(0) @RT(38)profile RPM reduce percentage (0-100%) @RT(0)
@END_Attrib
1 0 @F @F @F @F

@Var @RT(21)miMaxRPMDigitsToFloor @RT(0) @T @F @DT @RT(4)SINT @RT(0) @T @T @BASIC 0 @F
@F @F
@T
@BEG_Attrib
3 @RT(1)0 @RT(43)significant digits to floor for RPM profile @RT(0)
@END_Attrib
1 0 @F @F @F @F

@Var @RT(24)sv_iReadMachineDataCount @RT(0) @T @T @RENAMED 0 @T @T @DT @RT(5)UDINT @RT(0) @T @T @BASIC 0 @F
@F @F
@T
@BEG_Attrib
3 @RT(0) @RT(0) @RT(0)
@END_Attrib
1 8 @F @F @F @F

@END_Dcl

@END_Export

@BEG_Body

7

@BEG_Export

@BEG_Algo
@ALGORITHM @RT(16)aUpdateLintabOut @STRUCTURED_TEXT
@RT(0) @RT(0) @RT(0) @F @F
@END_Algo

@BEG_Dcl
@RT(16)DclTreeContainer
1
@Var @RT(1)i @RT(0) @T @F @DT @RT(5)UDINT @RT(0) @T @T @BASIC 0 @F
@F @F
@T
@BEG_Attrib
3 @RT(0) @RT(0) @RT(0)
@END_Attrib
1 4 @F @F @F @F

@END_Dcl

@END_Export

@BEG_Export

@BEG_Algo
@ALGORITHM @RT(13)aCalcMaxSpeed @STRUCTURED_TEXT
@RT(0) @RT(0) @RT(0) @F @F
@END_Algo

@BEG_Dcl
@RT(16)DclTreeContainer
0
@END_Dcl

@END_Export

@BEG_Export

@BEG_Algo
@ALGORITHM @RT(5)aInit @STRUCTURED_TEXT
@RT(0) @RT(0) @RT(0) @F @F
@END_Algo

@BEG_Dcl
@RT(16)DclTreeContainer
9
@Var @RT(15)prScrewDiameter @RT(0) @T @T @REFTO 0 @T @DT @RT(4)REAL @RT(0) @T @T @BASIC 0 @F
@F @F
@T
@BEG_Attrib
3 @RT(0) @RT(18)IN: screw diameter @RT(0)
@END_Attrib
1 1 @F @F @F @F

@Var @RT(8)prMaxRPM @RT(0) @T @T @REFTO 0 @T @DT @RT(4)REAL @RT(0) @T @T @BASIC 0 @F
@F @F
@T
@BEG_Attrib
3 @RT(0) @RT(20)IN: max RPM of screw @RT(0)
@END_Attrib
1 1 @F @F @F @F

@Var @RT(15)prMaxRPMProfile @RT(0) @T @T @REFTO 0 @T @DT @RT(4)REAL @RT(0) @T @T @BASIC 0 @F
@F @F
@T
@BEG_Attrib
3 @RT(0) @RT(28)IN: max RPM used for profile @RT(0)
@END_Attrib
1 1 @F @F @F @F

@Var @RT(21)prMaxRPMReducePercent @RT(0) @T @T @REFTO 0 @T @DT @RT(4)REAL @RT(0) @T @T @BASIC 0 @F
@F @F
@T
@BEG_Attrib
3 @RT(0) @RT(29)IN: max RPM reduce percentage @RT(0)
@END_Attrib
1 1 @F @F @F @F

@Var @RT(20)iMaxRPMDigitsToFloor @RT(0) @T @F @DT @RT(4)SINT @RT(0) @T @T @BASIC 0 @F
@F @F
@T
@BEG_Attrib
3 @RT(0) @RT(52)IN: max. significant digits to floor for RPM profile @RT(0)
@END_Attrib
1 1 @F @F @F @F

@Var @RT(10)pLintabInV @RT(0) @T @T @REFTO 0 @F @DERIVED 0 @T @T @DT @RT(16)KAPPL_LintabData @RT(0) @T @T @UNKNOWN 0 @F
@F @F
@T
@BEG_Attrib
3 @RT(0) @RT(25)IN: screw lintab RPM to % @RT(0)
@END_Attrib
1 1 @F @F @F @F

@Var @RT(11)pLintabOutV @RT(0) @T @T @REFTO 0 @F @DERIVED 0 @T @T @DT @RT(16)KAPPL_LintabData @RT(0) @T @T @UNKNOWN 0 @F
@F @F
@T
@BEG_Attrib
3 @RT(0) @RT(27)OUT: screw lintab cm/s to % @RT(0)
@END_Attrib
1 1 @F @F @F @F

@Var @RT(10)prMaxSpeed @RT(0) @T @T @REFTO 0 @T @DT @RT(4)REAL @RT(0) @T @T @BASIC 0 @F
@F @F
@T
@BEG_Attrib
3 @RT(0) @RT(43)OUT: max circumfence speed of screw in cm/s @RT(0)
@END_Attrib
1 1 @F @F @F @F

@Var @RT(3)tmp @RT(0) @T @F @DT @RT(4)DINT @RT(0) @T @T @BASIC 0 @F
@F @F
@T
@BEG_Attrib
3 @RT(0) @RT(0) @RT(0)
@END_Attrib
1 4 @F @F @F @F

@END_Dcl

@END_Export

@BEG_Export

@BEG_Algo
@POSTUPDATE_ALGORITHM @RT(10)pUpdateRPM @STRUCTURED_TEXT
@RT(0) @RT(10)mprMaxRPM^ @RT(9)PU_Task_7 @F @F
@END_Algo

@BEG_Dcl
@RT(16)DclTreeContainer
1
@Var @RT(13)rScalePercent @RT(0) @T @F @DT @RT(4)REAL @RT(0) @T @T @BASIC 0 @F
@F @F
@T
@BEG_Attrib
3 @RT(5)100.0 @RT(0) @RT(0)
@END_Attrib
1 0 @F @F @F @F

@END_Dcl

@END_Export

@BEG_Export

@BEG_Algo
@POSTUPDATE_ALGORITHM @RT(15)pUpdateVelocity @STRUCTURED_TEXT
@RT(0) @RT(35)mprScrewDiameter^,mprMaxRPMProfile^ @RT(9)PU_Task_7 @F @F
@END_Algo

@BEG_Dcl
@RT(16)DclTreeContainer
0
@END_Dcl

@END_Export

@BEG_Export

@BEG_Algo
@POSTUPDATE_ALGORITHM @RT(21)pUpdateVelocityLintab @STRUCTURED_TEXT
@RT(0) @RT(25)mprMaxSpeed^,mpLintabInV^ @RT(9)PU_Task_7 @F @F
@END_Algo

@BEG_Dcl
@RT(16)DclTreeContainer
0
@END_Dcl

@END_Export

@BEG_Export

@BEG_Algo
@POSTUPDATE_ALGORITHM @RT(18)pMachineDataLoaded @STRUCTURED_TEXT
@RT(0) @RT(24)sv_iReadMachineDataCount @RT(9)PU_Task_7 @F @F
@END_Algo

@BEG_Dcl
@RT(16)DclTreeContainer
0
@END_Dcl

@END_Export

@BEG_Body
@TL(12)
(**************************************** WARNING ********************************************
 *** The KEBA Kemro K2 System including software is not intended for safety control tasks! ***
 ***                       For further information see Comment tab!                        ***
 *********************************************************************************************)

(* convert lintab from RPM to cm/s screw circumfence speed *)
FOR i := 1 TO mpLintabInV^.LintabPoints.uNoOfPoints DO
   mpLintabOutV^.LintabPoints.Point[i].rX := FCalcScrewCircumfenceSpeed(rDiameter := mprScrewDiameter^, rRPM := mpLintabInV^.LintabPoints.Point[i].rX);// * rTmp;
   mpLintabOutV^.LintabPoints.Point[i].rY := mpLintabInV^.LintabPoints.Point[i].rY;
END_FOR;
mpLintabOutV^.LintabPoints.uNoOfPoints := mpLintabInV^.LintabPoints.uNoOfPoints;

@END_Body

@@@BEG_Comment@@@
@TL(0)

@@@END_Comment@@@

@BEG_Body
@TL(7)
(**************************************** WARNING ********************************************
 *** The KEBA Kemro K2 System including software is not intended for safety control tasks! ***
 ***                       For further information see Comment tab!                        ***
 *********************************************************************************************)

mprMaxSpeed^ := FCalcScrewCircumfenceSpeed(rDiameter := mprScrewDiameter^, rRPM := mprMaxRPMProfile^);

@END_Body

@@@BEG_Comment@@@
@TL(0)

@@@END_Comment@@@

@BEG_Body
@TL(60)
(**************************************** WARNING ********************************************
 *** The KEBA Kemro K2 System including software is not intended for safety control tasks! ***
 ***                       For further information see Comment tab!                        ***
 *********************************************************************************************)

mbInitDone := FALSE;

IF (NOT CHECK_REF(pLintabInV^)) OR (NOT CHECK_REF(pLintabOutV^)) THEN
    tmp := Print('pLintabInP or pLintabInV not valid');
    RETURN;
END_IF;

IF NOT CHECK_REF(prScrewDiameter^) THEN
    tmp := Print('prMaxPressure not valid');
    RETURN;
END_IF;

IF NOT CHECK_REF(prMaxRPM^) THEN
    tmp := Print('prMaxRPM not valid');
    RETURN;
END_IF;

IF NOT CHECK_REF(prMaxRPMProfile^) THEN
    tmp := Print('prMaxRPMProfile not valid');
    RETURN;
END_IF;

IF NOT CHECK_REF(prMaxRPMReducePercent^) THEN
    tmp := Print('prMaxRPMReducePercent not valid');
    RETURN;
END_IF;

IF NOT CHECK_REF(prMaxSpeed^) THEN
    tmp := Print('prMaxSpeed not valid');
    RETURN;
END_IF;

IF NOT CHECK_REF(prScrewDiameter^) THEN
    tmp := Print('prScrewDiameter not valid');
    RETURN;
END_IF;

mpLintabInV := pLintabInV;
mpLintabOutV := pLintabOutV;
mprScrewDiameter := prScrewDiameter;
mprMaxRPM := prMaxRPM;
mprMaxRPMProfile := prMaxRPMProfile;
mprMaxSpeed := prMaxSpeed;
mprMaxRPMReducePercent := prMaxRPMReducePercent;
miMaxRPMDigitsToFloor := iMaxRPMDigitsToFloor;

// init successful
mbInitDone := TRUE;

aCalcMaxSpeed();

aUpdateLintabOut();

@END_Body

@@@BEG_Comment@@@
@TL(7)
update pressure / speed lintabs for plast movement

update pLintabOutP and pLintabOutV according to the other parameters
the out lintab is updated when one of the input parameters changes
prMaxPressure points to the max pressure variable of the movement
prMaxSpeed is the maximum circumfence speed of the screw
it will be updated when max RPM input value or the prScrewDiameter changes
@@@END_Comment@@@

@BEG_Body
@TL(22)
(**************************************** WARNING ********************************************
 *** The KEBA Kemro K2 System including software is not intended for safety control tasks! ***
 ***                       For further information see Comment tab!                        ***
 *********************************************************************************************)

IF NOT mbInitDone OR (sv_DataState = nReadMachineData) THEN
   RETURN;
END_IF;

IF (sv_DataState = nReady AND (mprMaxRPMProfile^ > mprMaxRPM^)) THEN
   // prevent recalculation on machine data load except if max. value exceeds custom value
   IF mprMaxRPMReducePercent <> EMPTY THEN
      rScalePercent := 100.0 - mprMaxRPMReducePercent^;
   END_IF;
   mprMaxRPMProfile^ := FScaleAndFloor(mprMaxRPM^, rScalePercent, miMaxRPMDigitsToFloor);
END_IF;

@END_Body

@@@BEG_Comment@@@
@TL(0)

@@@END_Comment@@@

@BEG_Body
@TL(14)
(**************************************** WARNING ********************************************
 *** The KEBA Kemro K2 System including software is not intended for safety control tasks! ***
 ***                       For further information see Comment tab!                        ***
 *********************************************************************************************)

IF NOT mbInitDone OR (sv_DataState = nReadMachineData) THEN
   RETURN;
END_IF;

aCalcMaxSpeed();

@END_Body

@@@BEG_Comment@@@
@TL(0)

@@@END_Comment@@@

@BEG_Body
@TL(16)
(**************************************** WARNING ********************************************
 *** The KEBA Kemro K2 System including software is not intended for safety control tasks! ***
 ***                       For further information see Comment tab!                        ***
 *********************************************************************************************)

IF NOT mbInitDone THEN
    RETURN;
END_IF;

//update lintab
aUpdateLintabOut();

@END_Body

@@@BEG_Comment@@@
@TL(0)

@@@END_Comment@@@

@BEG_Body
@TL(7)
(**************************************** WARNING ********************************************
 *** The KEBA Kemro K2 System including software is not intended for safety control tasks! ***
 ***                       For further information see Comment tab!                        ***
 *********************************************************************************************)

aCalcMaxSpeed();

@END_Body

@@@BEG_Comment@@@
@TL(0)

@@@END_Comment@@@
@END_Body

@END_Contents
